// SIMATIC S7-200 SMART project (STEP 7-Micro/WIN SMART), CPU SR40

SYMBOL_TABLE 表格 1
阶段1计数器           C0
阶段2计数器           C1
阶段3计数器           C2
阶段4计数器           C3
阶段5计数器           C4
阶段6计数器           C5
分钟计数器_系统时间       C100
小时计数器_系统时间       C101
轮数计数器_系统时间       C102
通讯状态1            M0.1
通讯状态2            M0.2
本地启动CMD          M2.0
本地停止CMD          M2.1
本地复位CMD          M2.2
远程启动CMD          M3.0
远程停止CMD          M3.1
远程复位CMD          M3.2
PID故障码           MB20
通讯报错1            MB21
通讯报错2            MB22
吹扫时长定时器          T101
点火延时定时器          T102
升降档刷新时间          T103
点失败延时定时器         T104
主火阀开启延时计时器       T105
检漏0延时定时器         T110
检漏1延时定时器         T111
检漏2延时定时器         T112
检漏3延时定时器         T113
检漏4延时定时器         T114
空气阀检测定时器         T115
燃气阀检测定时器         T116
调节阀检测2定时器        T117
DCS安全联锁信号        V0.0
空气压力低检测          V0.1
燃气压力高检测          V0.2
燃气压力低检测          V0.3
JES258故障         V0.4
有火信号             V0.5
启动               V0.6
停止               V0.7
复位               V1.0
本地远程信号           V1.1
故障报警             V2.0
JES运行            V2.1
主火运行             V2.2
故障复位             V2.3
有火指示输出           V2.4
启动状态             V2.5
停止状态             V2.6
安全阀              V2.7
调节阀故障            V3.0
报警显示             V3.1
本地_远程            V20.0
升档               V20.1
降档               V20.2
自动手动             V20.3
PID自动            V20.5
吹扫动画显示           V20.7
无故障点火            V21.0
点火状态             V21.1
开始吹扫             V21.2
开始点火             V21.3
点火成功             V21.4
点火失败             V21.5
火焰信号丢失           V21.6
超温停机             V21.7
燃气阀反馈比对超限        V22.0
空气阀反馈比对超限        V22.1
DCS故障            V22.2
空气压力低            V22.3
燃气压力高            V22.4
燃气压力低            V22.5
空气调节阀故障1         V22.7
燃气调节阀故障          V23.0
调节阀点火位延时         V23.1
吹扫结束             V24.0
点火延时结束           V24.1
故障输出             V24.2
点火延时开始           V24.3
阶段一设定温度读值        V25.0
阶段二设定温度读值        V25.1
条件故障             M4.0
阶段三设定温度读值        V25.2
阶段四设定温度读值        V25.3
阶段五设定温度读值        V25.4
阶段六设定温度读值        V25.5
故障状态RTU          V620.0
自动状态RTU          V620.1
启动状态RTU          V620.2
停止状态RTU          V620.3
远程状态RTU          V620.4
远程启动             V620.5
远程停止             V620.6
远程复位             V620.7
远程升档             V621.0
远程降档             V621.1
当前温度R            VD304
温度显示             VD504
燃气显示             VD508
空气显示             VD512
温度上限设定值          VD520
温度下限设定值          VD524
超温停机设定值          VD528
燃气差              VD532
空气差              VD536
燃气给定             VD540
空气给定             VD544
燃气偏差允许值          VD548
空气偏差允许值          VD552
吹扫空气阀开度          VD564
PID设定温度          VD568
PID微分_D          VD572
PID增益_P          VD576
PID积分_I          VD580
PID采样时间          VD584
PID手动值           VD588
吹扫计时开始_值         VD592
PID档位D           VD596
当前档位显示           VD600
档位设置             VD604
当量_每档            VD608
PID输出换算档位        VD612
PID档位R           VD616
空气               VD640
燃气               VD644
温度               VD648
当前档位             VD652
燃气1档_0档          VD700
燃气2档_点火档         VD704
燃气3档_1档          VD708
燃气4档             VD712
燃气5档             VD716
燃气6档             VD720
燃气7档             VD724
燃气8档             VD728
燃气9档             VD732
燃气10档            VD736
燃气11档            VD740
燃气12档            VD744
燃气13档            VD748
燃气14档            VD752
燃气15档            VD756
燃气16档            VD760
燃气17档            VD764
燃气18档            VD768
燃气19档            VD772
燃气20档            VD776
空气1档             VD780
空气2档             VD784
空气3档             VD788
空气4档             VD792
空气5档             VD796
空气6档             VD800
空气7档             VD804
空气8档             VD808
空气9档             VD812
空气10档            VD816
空气11档            VD820
空气12档            VD824
空气13档            VD828
空气14档            VD832
空气15档            VD836
空气16档            VD840
空气17档            VD844
空气18档            VD848
空气19档            VD852
空气20档            VD856
阶段1温度            VD860
阶段2温度            VD864
阶段3温度            VD868
阶段4温度            VD872
阶段5温度            VD876
阶段6温度            VD880
吹扫时间设定           VW200
点火延时设定值          VW202
吹扫延时             VW206
主火阀开启延时          VW208
PID输出            VW210
阶段1              VW220
阶段2              VW222
阶段3              VW224
阶段4              VW226
阶段5              VW228
阶段6              VW230
阶段1设定            VW232
阶段2设定            VW234
阶段3设定            VW236
阶段4设定            VW238
阶段5设定            VW240
阶段6设定            VW242
调节阀检测延时          VW244
当前温度             VW898
END_SYMBOL_TABLE

SYMBOL_TABLE 系统符号
Always_On        SM0.0    // 始终接通
First_Scan_On    SM0.1    // 仅在第一个扫描周期时接通
Clock_60s        SM0.4    // 针对 1 分钟的周期时间，时钟脉冲接通 30 s，断开 30 s.
Clock_1s         SM0.5    // 针对 1 s 的周期时间，时钟脉冲接通 0.5 s，断开 0.5 s.
END_SYMBOL_TABLE

SYMBOL_TABLE 检漏符号表
检漏标志             VB41     // 0:停止检漏 1:检漏中 2:检漏完成
检漏程序步            VB40     // 检漏第1、2、3、4步
大火指示             V31.0
检漏通过             V30.6
检漏异常2            V30.5
检漏异常1            V30.4
阀1_2             V30.3
阀2_2             V30.2
阀1_1             V30.1
阀2_1             V30.0
检漏异常             V22.6
END_SYMBOL_TABLE

ORGANIZATION_BLOCK 程序块:OB1
TITLE=程序注释
BEGIN
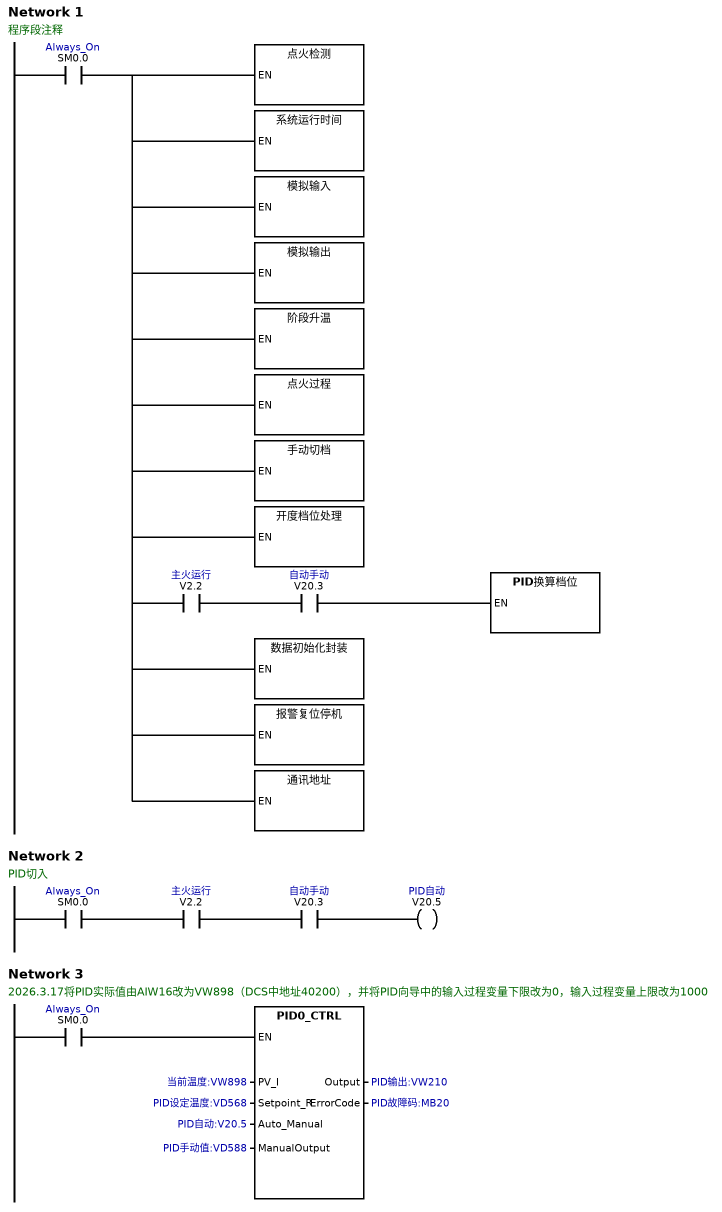
Network 1
// 程序段注释
LD     Always_On:SM0.0
LPS
CALL   点火检测:SBR4
CALL   系统运行时间:SBR5
CALL   模拟输入:SBR0
CALL   模拟输出:SBR3
CALL   阶段升温:SBR6
CALL   点火过程:SBR8
CALL   手动切档:SBR11
CALL   开度档位处理:SBR12
A      主火运行:V2.2
A      自动手动:V20.3
CALL   PID换算档位:SBR13
LRD
CALL   数据初始化封装:SBR14
LRD
CALL   报警复位停机:SBR16
LPP
CALL   通讯地址:SBR19
Network 2
// PID切入
LD     Always_On:SM0.0
A      主火运行:V2.2
A      自动手动:V20.3
=      PID自动:V20.5
Network 3
// 2026.3.17将PID实际值由AIW16改为VW898（DCS中地址40200），并将PID向导中的输入过程变量下限改为0，输入过程变量上限改为1000
LD     Always_On:SM0.0
CALL   PID0_CTRL:SBR18, 当前温度:VW898, PID设定温度:VD568, PID自动:V20.5, PID手动值:VD588, PID输出:VW210, PID故障码:MB20
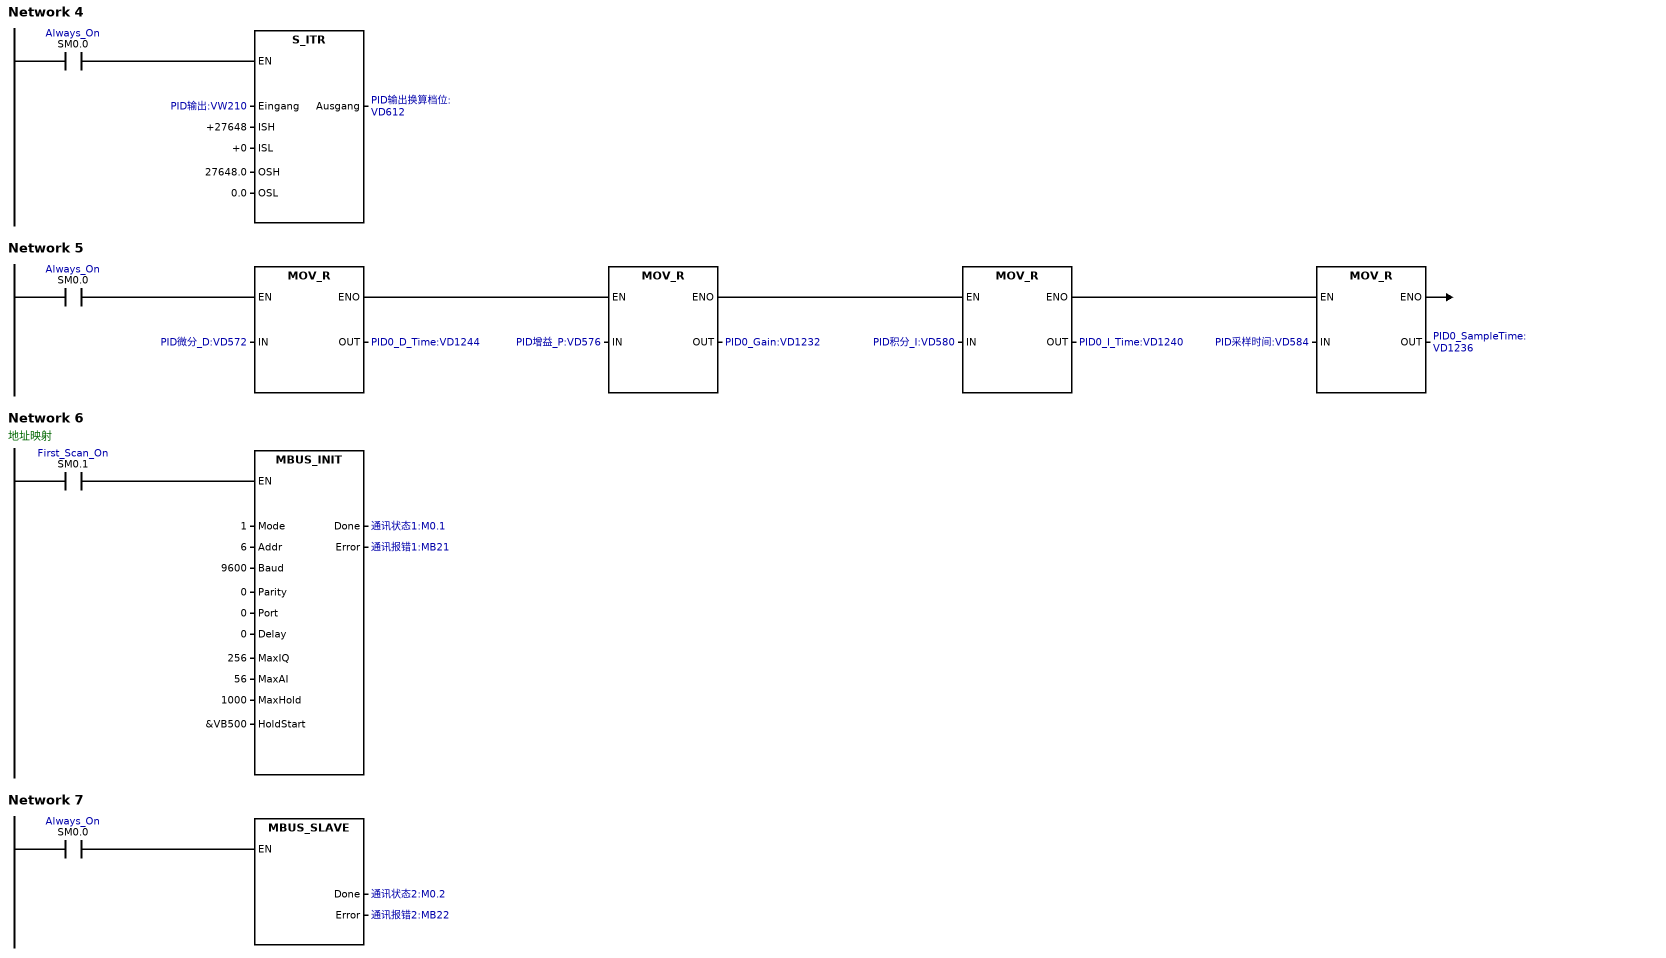
Network 4
LD     Always_On:SM0.0
CALL   S_ITR:SBR1, PID输出:VW210, +27648, +0, 27648.0, 0.0, PID输出换算档位:VD612
Network 5
LD     Always_On:SM0.0
MOVR   PID微分_D:VD572, PID0_D_Time:VD1244
AENO
MOVR   PID增益_P:VD576, PID0_Gain:VD1232
AENO
MOVR   PID积分_I:VD580, PID0_I_Time:VD1240
AENO
MOVR   PID采样时间:VD584, PID0_SampleTime:VD1236
Network 6
// 地址映射
LD     First_Scan_On:SM0.1
CALL   MBUS_INIT:SBR7, 1, 6, 9600, 0, 0, 0, 256, 56, 1000, &VB500, 通讯状态1:M0.1, 通讯报错1:MB21
Network 7
LD     Always_On:SM0.0
CALL   MBUS_SLAVE:SBR9, 通讯状态2:M0.2, 通讯报错2:MB22
END_ORGANIZATION_BLOCK

SUBROUTINE_BLOCK 模拟输入:SBR0
TITLE=子程序注释
BEGIN
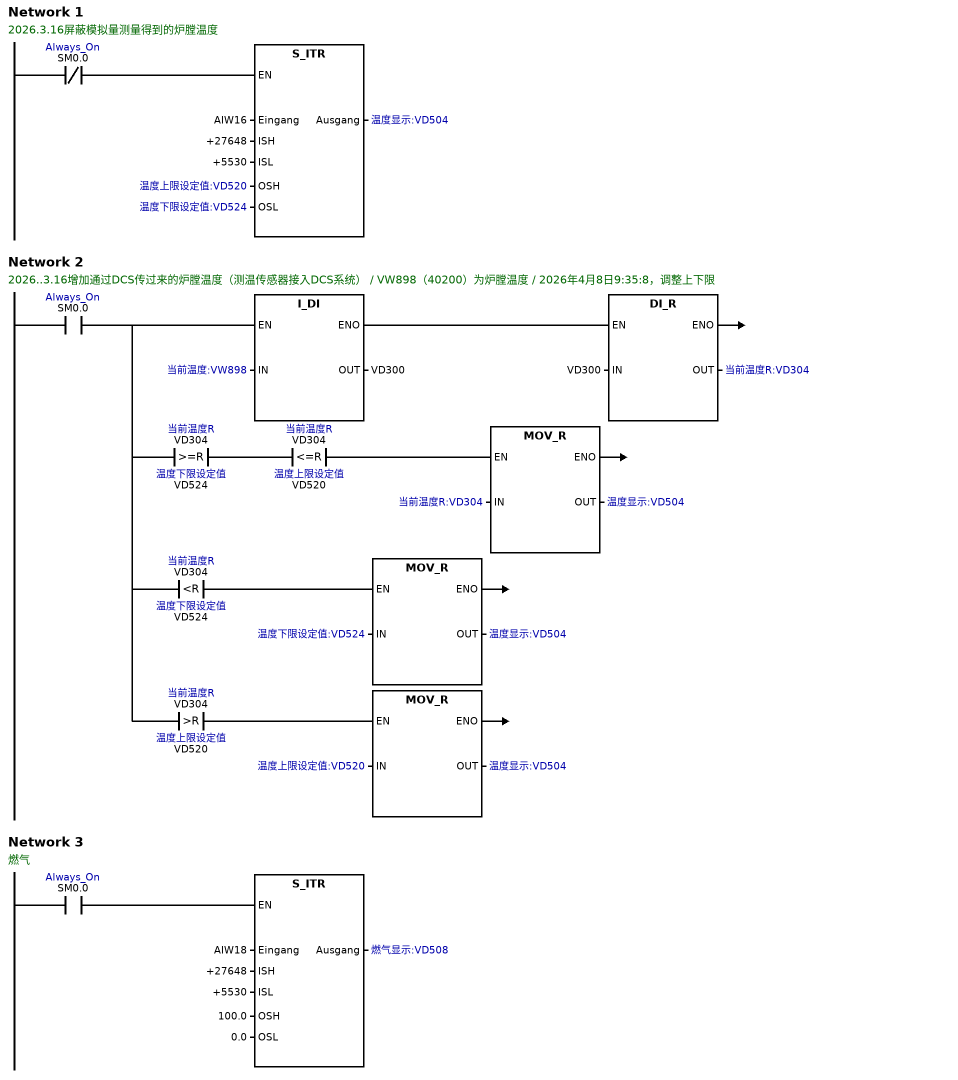
Network 1
// 2026.3.16屏蔽模拟量测量得到的炉膛温度
LDN    Always_On:SM0.0
CALL   S_ITR:SBR1, AIW16, +27648, +5530, 温度上限设定值:VD520, 温度下限设定值:VD524, 温度显示:VD504
Network 2
// 2026..3.16增加通过DCS传过来的炉膛温度（测温传感器接入DCS系统）
// VW898（40200）为炉膛温度
// 2026年4月8日9:35:8，调整上下限
LD     Always_On:SM0.0
LPS
ITD    当前温度:VW898, VD300
AENO
DTR    VD300, 当前温度R:VD304
LRD
AR>=   当前温度R:VD304, 温度下限设定值:VD524
AR<=   当前温度R:VD304, 温度上限设定值:VD520
MOVR   当前温度R:VD304, 温度显示:VD504
LRD
AR<    当前温度R:VD304, 温度下限设定值:VD524
MOVR   温度下限设定值:VD524, 温度显示:VD504
LPP
AR>    当前温度R:VD304, 温度上限设定值:VD520
MOVR   温度上限设定值:VD520, 温度显示:VD504
Network 3
// 燃气
LD     Always_On:SM0.0
CALL   S_ITR:SBR1, AIW18, +27648, +5530, 100.0, 0.0, 燃气显示:VD508
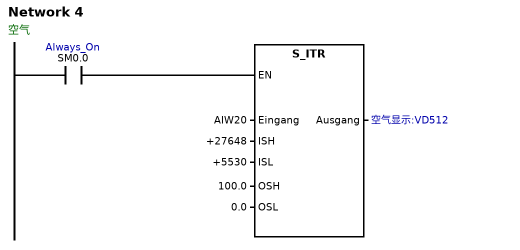
Network 4
// 空气
LD     Always_On:SM0.0
CALL   S_ITR:SBR1, AIW20, +27648, +5530, 100.0, 0.0, 空气显示:VD512
END_SUBROUTINE_BLOCK

// SBR1: protected block, not included

// SBR2: protected block, not included

SUBROUTINE_BLOCK 模拟输出:SBR3
TITLE=
BEGIN
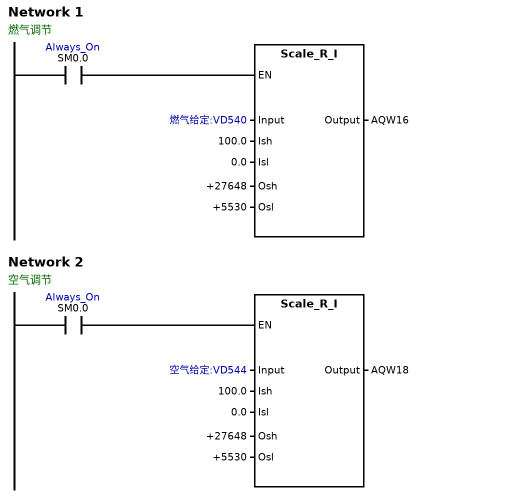
Network 1
// 燃气调节
LD     Always_On:SM0.0
CALL   Scale_R_I:SBR17, 燃气给定:VD540, 100.0, 0.0, +27648, +5530, AQW16
Network 2
// 空气调节
LD     Always_On:SM0.0
CALL   Scale_R_I:SBR17, 空气给定:VD544, 100.0, 0.0, +27648, +5530, AQW18
END_SUBROUTINE_BLOCK

SUBROUTINE_BLOCK 点火检测:SBR4
TITLE=
BEGIN
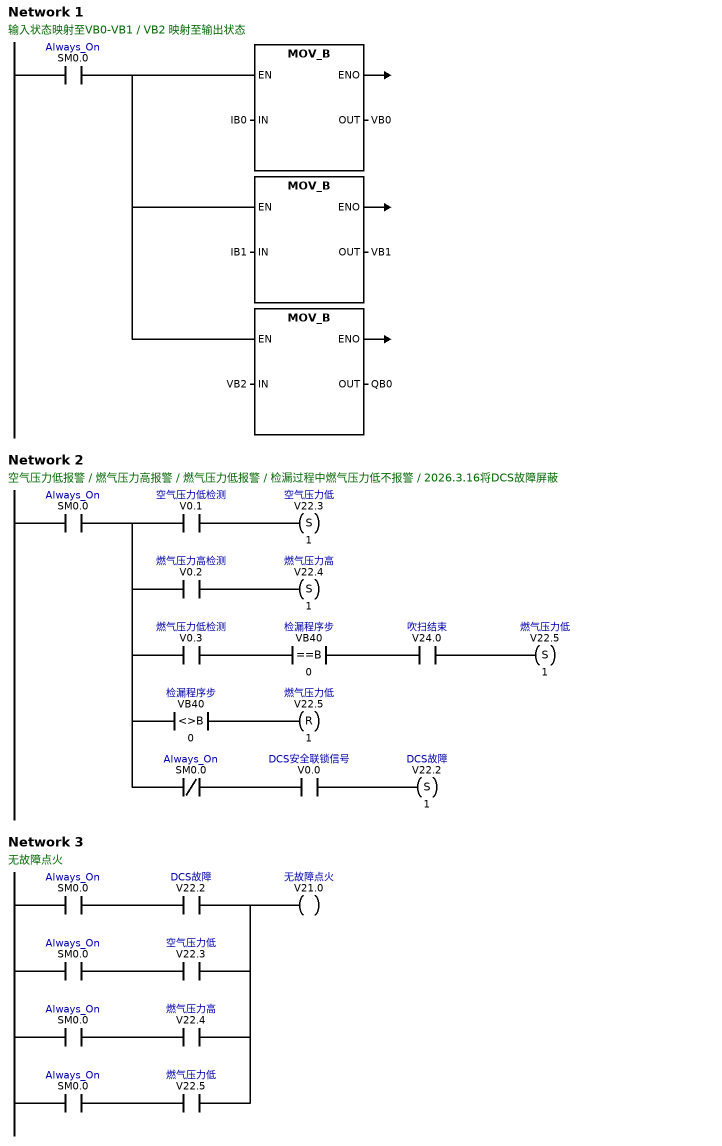
Network 1
// 输入状态映射至VB0-VB1
// VB2 映射至输出状态
LD     Always_On:SM0.0
MOVB   IB0, VB0
MOVB   IB1, VB1
MOVB   VB2, QB0
Network 2
// 空气压力低报警
// 燃气压力高报警
// 燃气压力低报警
// 检漏过程中燃气压力低不报警
// 2026.3.16将DCS故障屏蔽
LD     Always_On:SM0.0
LPS
A      空气压力低检测:V0.1
S      空气压力低:V22.3, 1
LRD
A      燃气压力高检测:V0.2
S      燃气压力高:V22.4, 1
LRD
A      燃气压力低检测:V0.3
AB=    检漏程序步:VB40, 0
A      吹扫结束:V24.0
S      燃气压力低:V22.5, 1
LRD
AB<>   检漏程序步:VB40, 0
R      燃气压力低:V22.5, 1
LPP
AN     Always_On:SM0.0
A      DCS安全联锁信号:V0.0
S      DCS故障:V22.2, 1
Network 3
// 无故障点火
LD     Always_On:SM0.0
A      DCS故障:V22.2
LD     Always_On:SM0.0
A      空气压力低:V22.3
OLD
LD     Always_On:SM0.0
A      燃气压力高:V22.4
OLD
LD     Always_On:SM0.0
A      燃气压力低:V22.5
OLD
=      无故障点火:V21.0
END_SUBROUTINE_BLOCK

SUBROUTINE_BLOCK 系统运行时间:SBR5
TITLE=
BEGIN
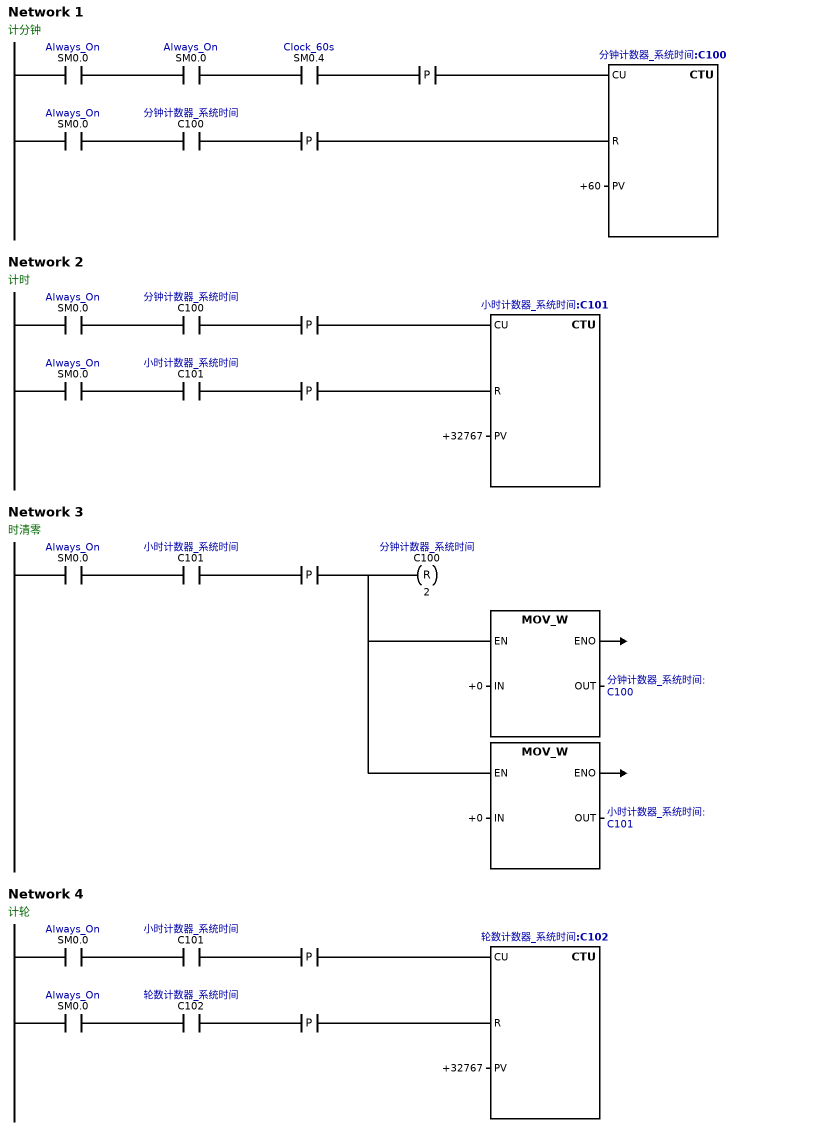
Network 1
// 计分钟
LD     Always_On:SM0.0
A      Always_On:SM0.0
A      Clock_60s:SM0.4
EU
LD     Always_On:SM0.0
A      分钟计数器_系统时间:C100
EU
CTU    分钟计数器_系统时间:C100, +60
Network 2
// 计时
LD     Always_On:SM0.0
A      分钟计数器_系统时间:C100
EU
LD     Always_On:SM0.0
A      小时计数器_系统时间:C101
EU
CTU    小时计数器_系统时间:C101, +32767
Network 3
// 时清零
LD     Always_On:SM0.0
A      小时计数器_系统时间:C101
EU
R      分钟计数器_系统时间:C100, 2
MOVW   +0, 分钟计数器_系统时间:C100
MOVW   +0, 小时计数器_系统时间:C101
Network 4
// 计轮
LD     Always_On:SM0.0
A      小时计数器_系统时间:C101
EU
LD     Always_On:SM0.0
A      轮数计数器_系统时间:C102
EU
CTU    轮数计数器_系统时间:C102, +32767
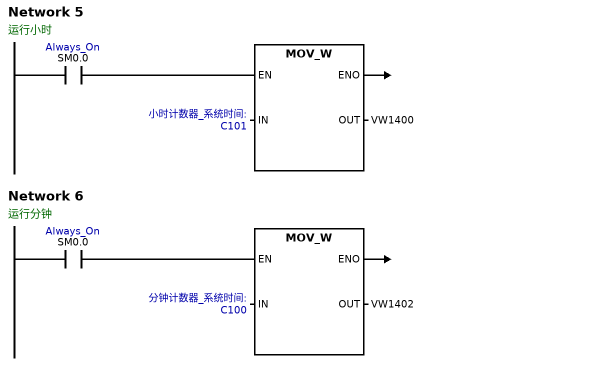
Network 5
// 运行小时
LD     Always_On:SM0.0
MOVW   小时计数器_系统时间:C101, VW1400
Network 6
// 运行分钟
LD     Always_On:SM0.0
MOVW   分钟计数器_系统时间:C100, VW1402
END_SUBROUTINE_BLOCK

SUBROUTINE_BLOCK 阶段升温:SBR6
TITLE=
BEGIN
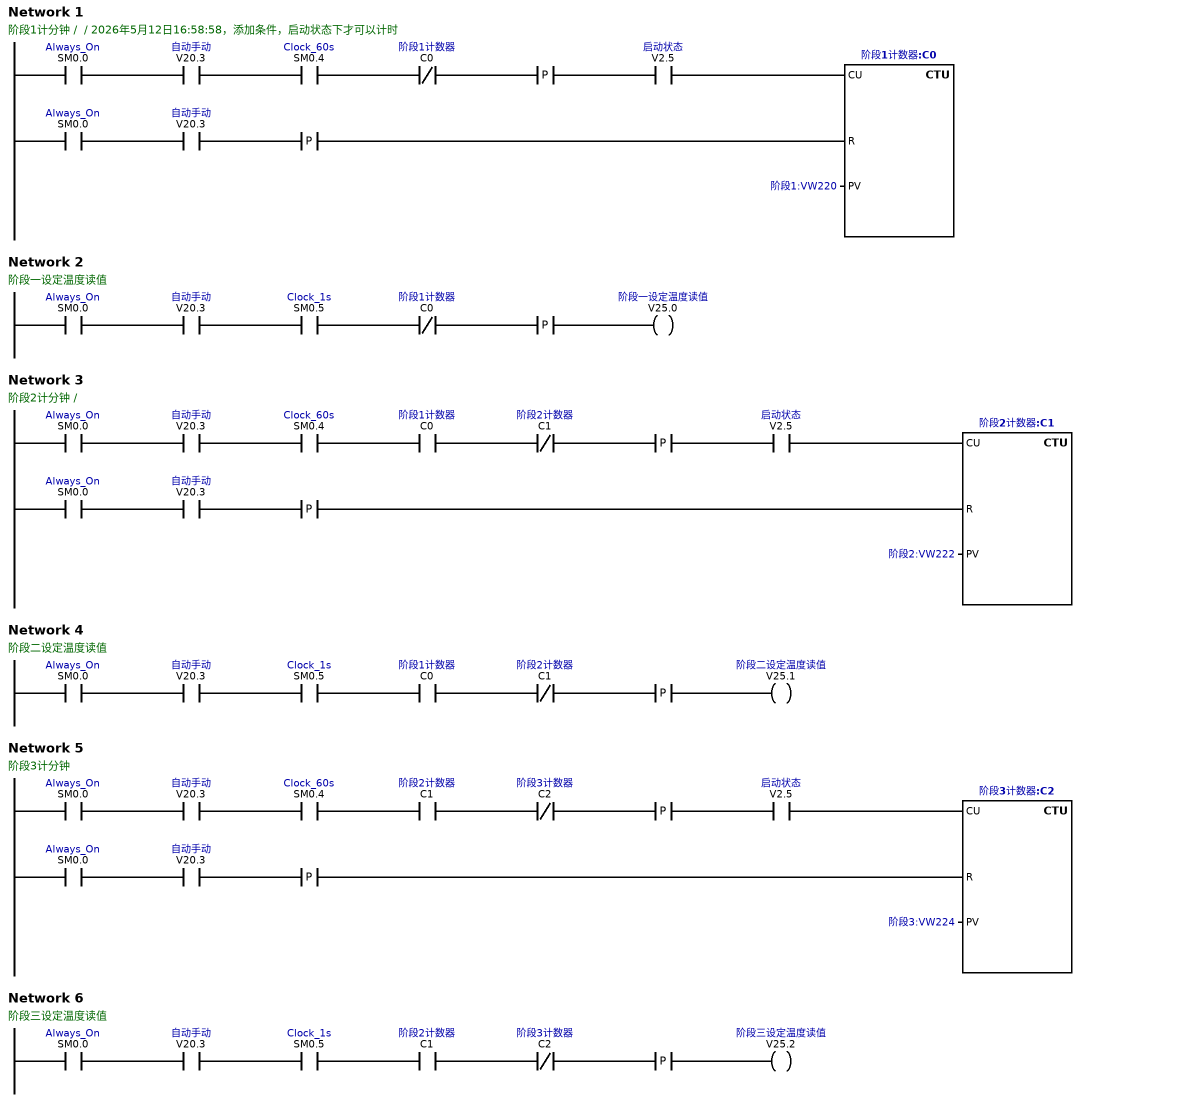
Network 1
// 阶段1计分钟
// 
// 2026年5月12日16:58:58，添加条件，启动状态下才可以计时
LD     Always_On:SM0.0
A      自动手动:V20.3
A      Clock_60s:SM0.4
AN     阶段1计数器:C0
EU
A      启动状态:V2.5
LD     Always_On:SM0.0
A      自动手动:V20.3
EU
CTU    阶段1计数器:C0, 阶段1:VW220
Network 2
// 阶段一设定温度读值
LD     Always_On:SM0.0
A      自动手动:V20.3
A      Clock_1s:SM0.5
AN     阶段1计数器:C0
EU
=      阶段一设定温度读值:V25.0
Network 3
// 阶段2计分钟
// 
LD     Always_On:SM0.0
A      自动手动:V20.3
A      Clock_60s:SM0.4
A      阶段1计数器:C0
AN     阶段2计数器:C1
EU
A      启动状态:V2.5
LD     Always_On:SM0.0
A      自动手动:V20.3
EU
CTU    阶段2计数器:C1, 阶段2:VW222
Network 4
// 阶段二设定温度读值
LD     Always_On:SM0.0
A      自动手动:V20.3
A      Clock_1s:SM0.5
A      阶段1计数器:C0
AN     阶段2计数器:C1
EU
=      阶段二设定温度读值:V25.1
Network 5
// 阶段3计分钟
LD     Always_On:SM0.0
A      自动手动:V20.3
A      Clock_60s:SM0.4
A      阶段2计数器:C1
AN     阶段3计数器:C2
EU
A      启动状态:V2.5
LD     Always_On:SM0.0
A      自动手动:V20.3
EU
CTU    阶段3计数器:C2, 阶段3:VW224
Network 6
// 阶段三设定温度读值
LD     Always_On:SM0.0
A      自动手动:V20.3
A      Clock_1s:SM0.5
A      阶段2计数器:C1
AN     阶段3计数器:C2
EU
=      阶段三设定温度读值:V25.2
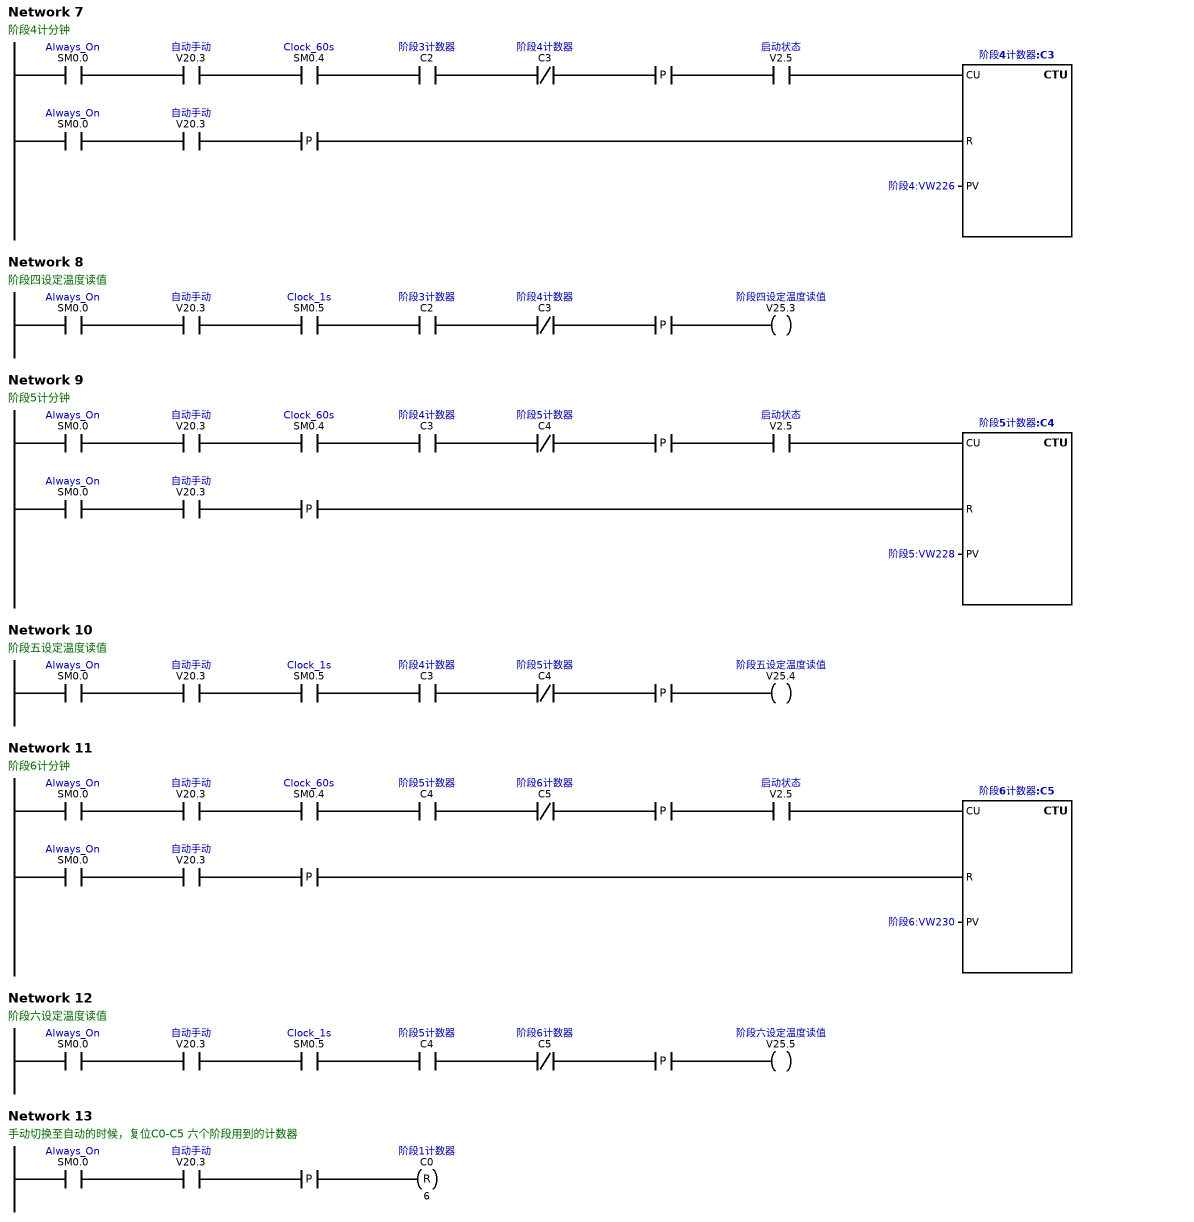
Network 7
// 阶段4计分钟
LD     Always_On:SM0.0
A      自动手动:V20.3
A      Clock_60s:SM0.4
A      阶段3计数器:C2
AN     阶段4计数器:C3
EU
A      启动状态:V2.5
LD     Always_On:SM0.0
A      自动手动:V20.3
EU
CTU    阶段4计数器:C3, 阶段4:VW226
Network 8
// 阶段四设定温度读值
LD     Always_On:SM0.0
A      自动手动:V20.3
A      Clock_1s:SM0.5
A      阶段3计数器:C2
AN     阶段4计数器:C3
EU
=      阶段四设定温度读值:V25.3
Network 9
// 阶段5计分钟
LD     Always_On:SM0.0
A      自动手动:V20.3
A      Clock_60s:SM0.4
A      阶段4计数器:C3
AN     阶段5计数器:C4
EU
A      启动状态:V2.5
LD     Always_On:SM0.0
A      自动手动:V20.3
EU
CTU    阶段5计数器:C4, 阶段5:VW228
Network 10
// 阶段五设定温度读值
LD     Always_On:SM0.0
A      自动手动:V20.3
A      Clock_1s:SM0.5
A      阶段4计数器:C3
AN     阶段5计数器:C4
EU
=      阶段五设定温度读值:V25.4
Network 11
// 阶段6计分钟
LD     Always_On:SM0.0
A      自动手动:V20.3
A      Clock_60s:SM0.4
A      阶段5计数器:C4
AN     阶段6计数器:C5
EU
A      启动状态:V2.5
LD     Always_On:SM0.0
A      自动手动:V20.3
EU
CTU    阶段6计数器:C5, 阶段6:VW230
Network 12
// 阶段六设定温度读值
LD     Always_On:SM0.0
A      自动手动:V20.3
A      Clock_1s:SM0.5
A      阶段5计数器:C4
AN     阶段6计数器:C5
EU
=      阶段六设定温度读值:V25.5
Network 13
// 手动切换至自动的时候，复位C0-C5 六个阶段用到的计数器
LD     Always_On:SM0.0
A      自动手动:V20.3
EU
R      阶段1计数器:C0, 6
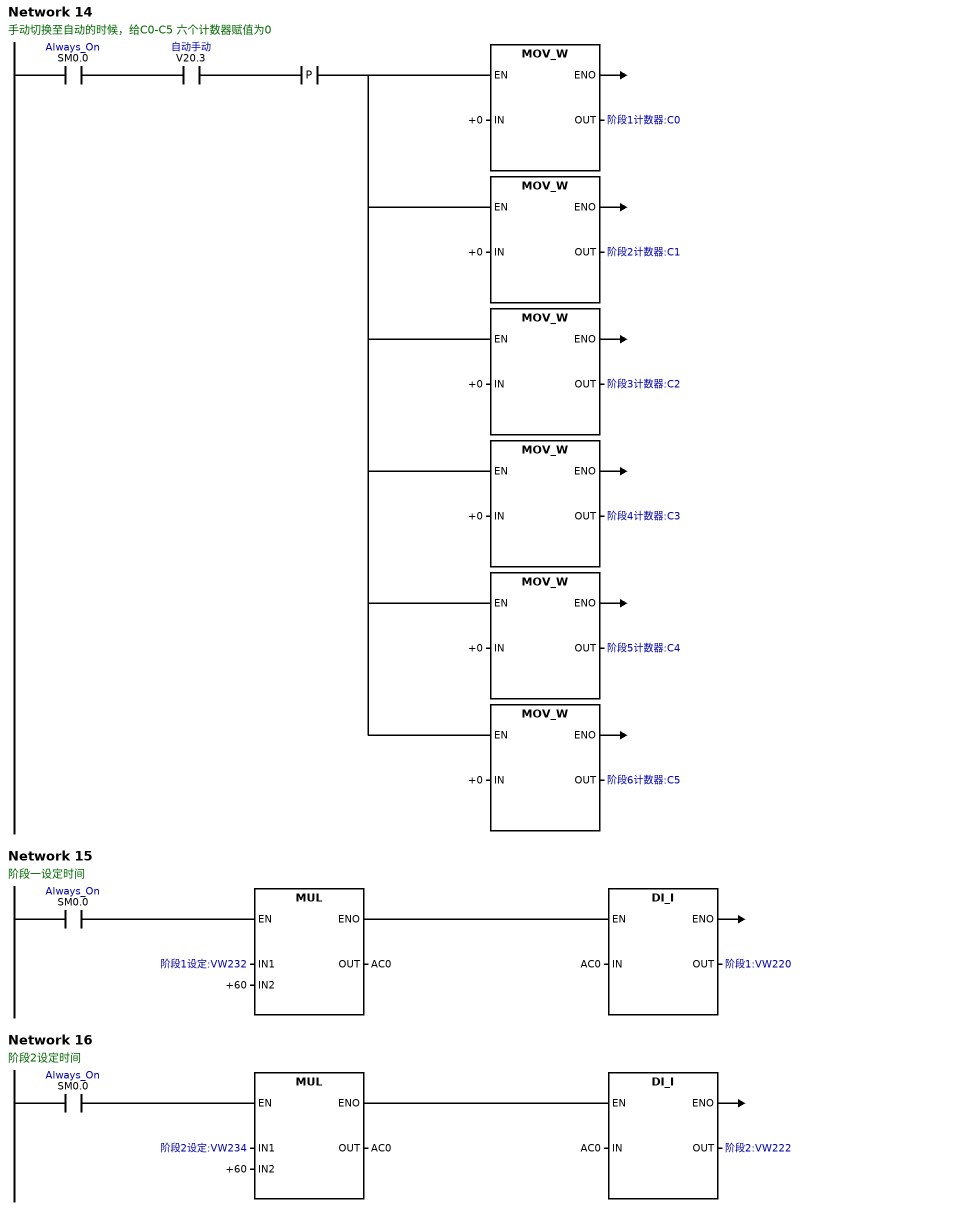
Network 14
// 手动切换至自动的时候，给C0-C5 六个计数器赋值为0
LD     Always_On:SM0.0
A      自动手动:V20.3
EU
MOVW   +0, 阶段1计数器:C0
MOVW   +0, 阶段2计数器:C1
MOVW   +0, 阶段3计数器:C2
MOVW   +0, 阶段4计数器:C3
MOVW   +0, 阶段5计数器:C4
MOVW   +0, 阶段6计数器:C5
Network 15
// 阶段一设定时间
LD     Always_On:SM0.0
MOVW   阶段1设定:VW232, AC0
AENO
MUL    +60, AC0
AENO
DTI    AC0, 阶段1:VW220
Network 16
// 阶段2设定时间
LD     Always_On:SM0.0
MOVW   阶段2设定:VW234, AC0
AENO
MUL    +60, AC0
AENO
DTI    AC0, 阶段2:VW222
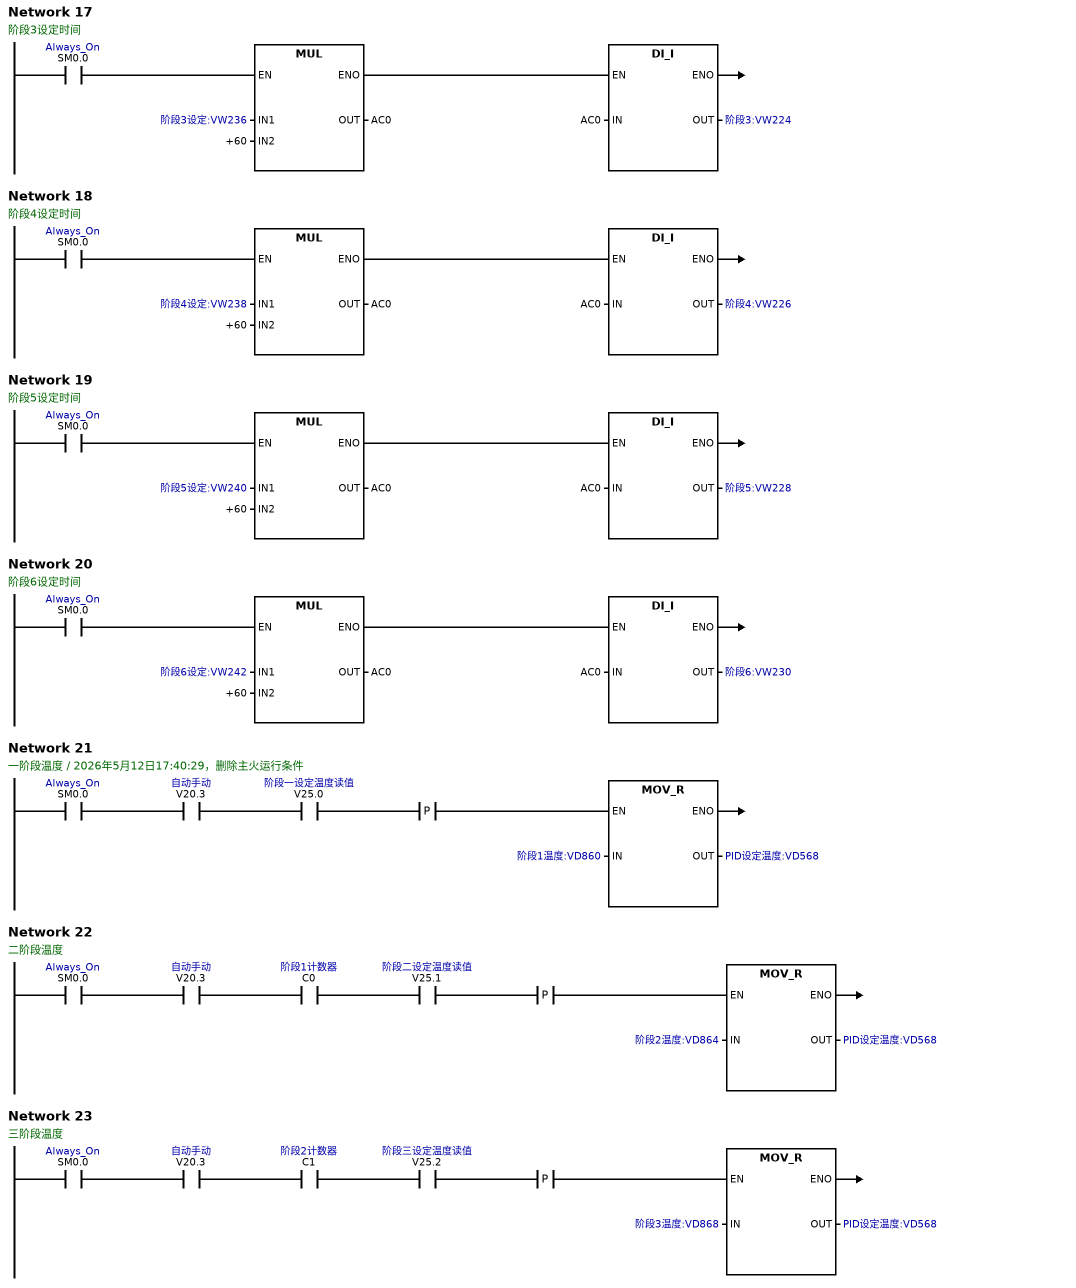
Network 17
// 阶段3设定时间
LD     Always_On:SM0.0
MOVW   阶段3设定:VW236, AC0
AENO
MUL    +60, AC0
AENO
DTI    AC0, 阶段3:VW224
Network 18
// 阶段4设定时间
LD     Always_On:SM0.0
MOVW   阶段4设定:VW238, AC0
AENO
MUL    +60, AC0
AENO
DTI    AC0, 阶段4:VW226
Network 19
// 阶段5设定时间
LD     Always_On:SM0.0
MOVW   阶段5设定:VW240, AC0
AENO
MUL    +60, AC0
AENO
DTI    AC0, 阶段5:VW228
Network 20
// 阶段6设定时间
LD     Always_On:SM0.0
MOVW   阶段6设定:VW242, AC0
AENO
MUL    +60, AC0
AENO
DTI    AC0, 阶段6:VW230
Network 21
// 一阶段温度
// 2026年5月12日17:40:29，删除主火运行条件
LD     Always_On:SM0.0
A      自动手动:V20.3
A      阶段一设定温度读值:V25.0
EU
MOVR   阶段1温度:VD860, PID设定温度:VD568
Network 22
// 二阶段温度
LD     Always_On:SM0.0
A      自动手动:V20.3
A      阶段1计数器:C0
A      阶段二设定温度读值:V25.1
EU
MOVR   阶段2温度:VD864, PID设定温度:VD568
Network 23
// 三阶段温度
LD     Always_On:SM0.0
A      自动手动:V20.3
A      阶段2计数器:C1
A      阶段三设定温度读值:V25.2
EU
MOVR   阶段3温度:VD868, PID设定温度:VD568
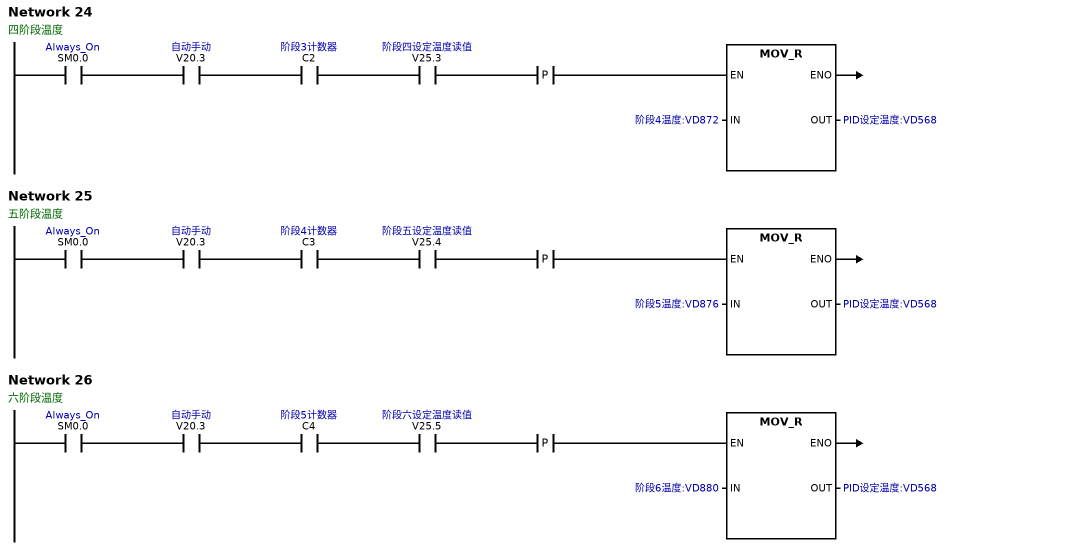
Network 24
// 四阶段温度
LD     Always_On:SM0.0
A      自动手动:V20.3
A      阶段3计数器:C2
A      阶段四设定温度读值:V25.3
EU
MOVR   阶段4温度:VD872, PID设定温度:VD568
Network 25
// 五阶段温度
LD     Always_On:SM0.0
A      自动手动:V20.3
A      阶段4计数器:C3
A      阶段五设定温度读值:V25.4
EU
MOVR   阶段5温度:VD876, PID设定温度:VD568
Network 26
// 六阶段温度
LD     Always_On:SM0.0
A      自动手动:V20.3
A      阶段5计数器:C4
A      阶段六设定温度读值:V25.5
EU
MOVR   阶段6温度:VD880, PID设定温度:VD568
END_SUBROUTINE_BLOCK

// SBR7: protected block, not included

SUBROUTINE_BLOCK 点火过程:SBR8
TITLE=
BEGIN
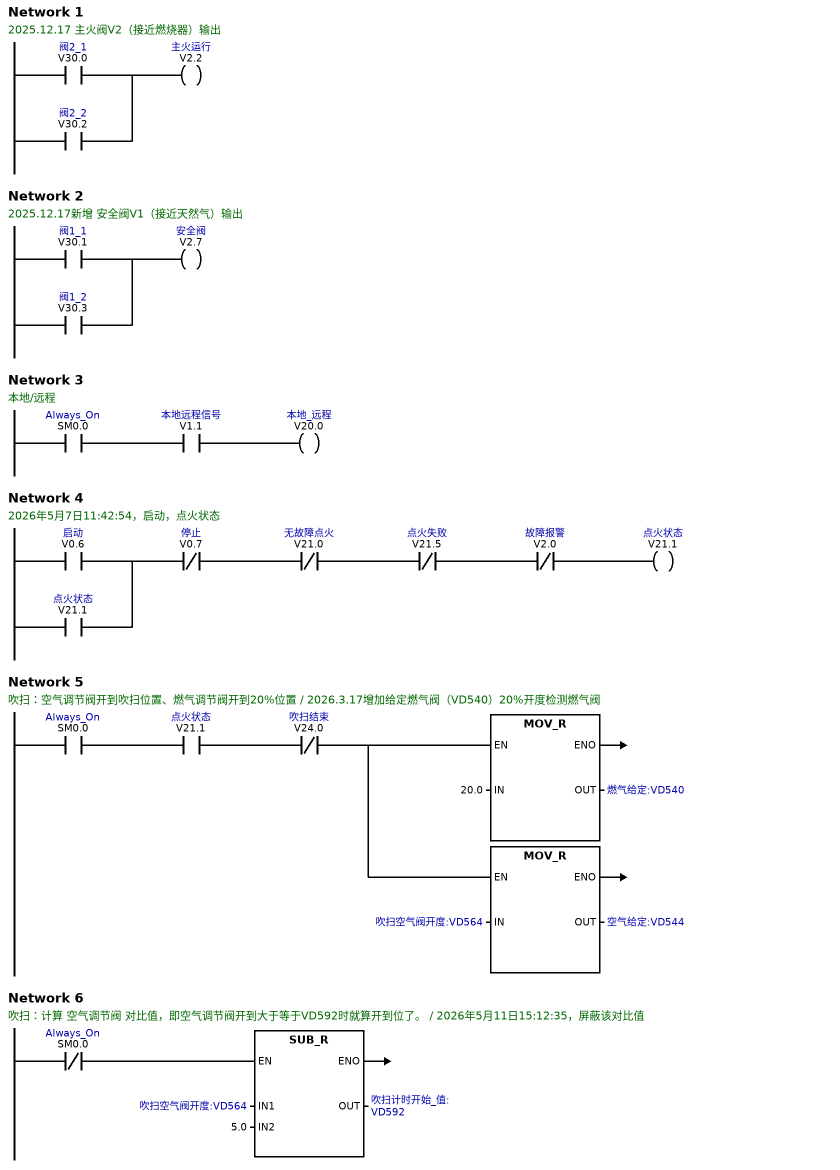
Network 1
// 2025.12.17 主火阀V2（接近燃烧器）输出
LD     阀2_1:V30.0
O      阀2_2:V30.2
=      主火运行:V2.2
Network 2
// 2025.12.17新增 安全阀V1（接近天然气）输出
LD     阀1_1:V30.1
O      阀1_2:V30.3
=      安全阀:V2.7
Network 3
// 本地/远程
LD     Always_On:SM0.0
A      本地远程信号:V1.1
=      本地_远程:V20.0
Network 4
// 2026年5月7日11:42:54，启动，点火状态
LD     启动:V0.6
O      点火状态:V21.1
AN     停止:V0.7
AN     无故障点火:V21.0
AN     点火失败:V21.5
AN     故障报警:V2.0
=      点火状态:V21.1
Network 5
// 吹扫：空气调节阀开到吹扫位置、燃气调节阀开到20%位置
// 2026.3.17增加给定燃气阀（VD540）20%开度检测燃气阀
LD     Always_On:SM0.0
A      点火状态:V21.1
AN     吹扫结束:V24.0
MOVR   20.0, 燃气给定:VD540
MOVR   吹扫空气阀开度:VD564, 空气给定:VD544
Network 6
// 吹扫：计算 空气调节阀 对比值，即空气调节阀开到大于等于VD592时就算开到位了。
// 2026年5月11日15:12:35，屏蔽该对比值
LDN    Always_On:SM0.0
MOVR   吹扫空气阀开度:VD564, 吹扫计时开始_值:VD592
-R     5.0, 吹扫计时开始_值:VD592
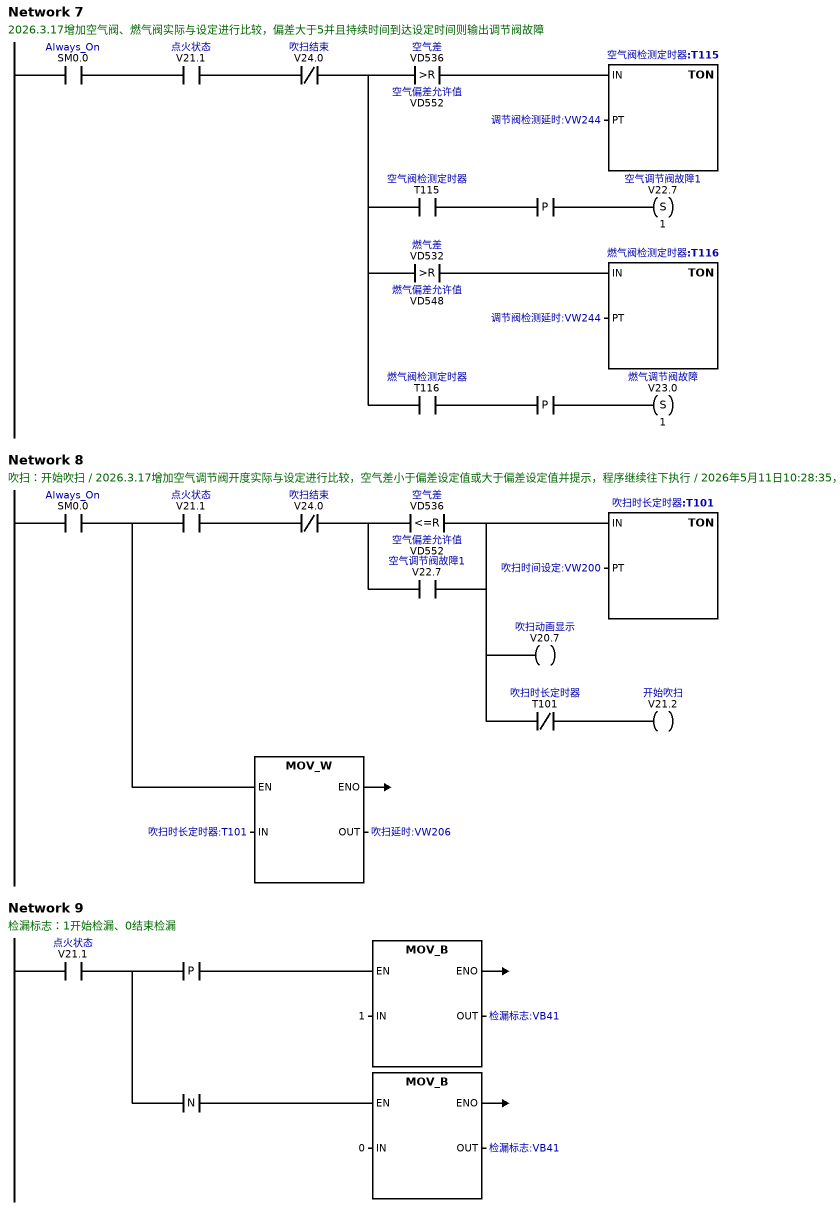
Network 7
// 2026.3.17增加空气阀、燃气阀实际与设定进行比较，偏差大于5并且持续时间到达设定时间则输出调节阀故障
LD     Always_On:SM0.0
A      点火状态:V21.1
AN     吹扫结束:V24.0
LPS
AR>    空气差:VD536, 空气偏差允许值:VD552
TON    空气阀检测定时器:T115, 调节阀检测延时:VW244
LRD
A      空气阀检测定时器:T115
EU
S      空气调节阀故障1:V22.7, 1
LRD
AR>    燃气差:VD532, 燃气偏差允许值:VD548
TON    燃气阀检测定时器:T116, 调节阀检测延时:VW244
LPP
A      燃气阀检测定时器:T116
EU
S      燃气调节阀故障:V23.0, 1
Network 8
// 吹扫：开始吹扫
// 2026.3.17增加空气调节阀开度实际与设定进行比较，空气差小于偏差设定值或大于偏差设定值并提示，程序继续往下执行
// 2026年5月11日10:28:35，显示吹扫时长
LD     Always_On:SM0.0
LPS
A      点火状态:V21.1
AN     吹扫结束:V24.0
LDR<=  空气差:VD536, 空气偏差允许值:VD552
O      空气调节阀故障1:V22.7
ALD
TON    吹扫时长定时器:T101, 吹扫时间设定:VW200
=      吹扫动画显示:V20.7
AN     吹扫时长定时器:T101
=      开始吹扫:V21.2
LPP
MOVW   吹扫时长定时器:T101, 吹扫延时:VW206
Network 9
// 检漏标志：1开始检漏、0结束检漏
LD     点火状态:V21.1
LPS
EU
MOVB   1, 检漏标志:VB41
LPP
ED
MOVB   0, 检漏标志:VB41
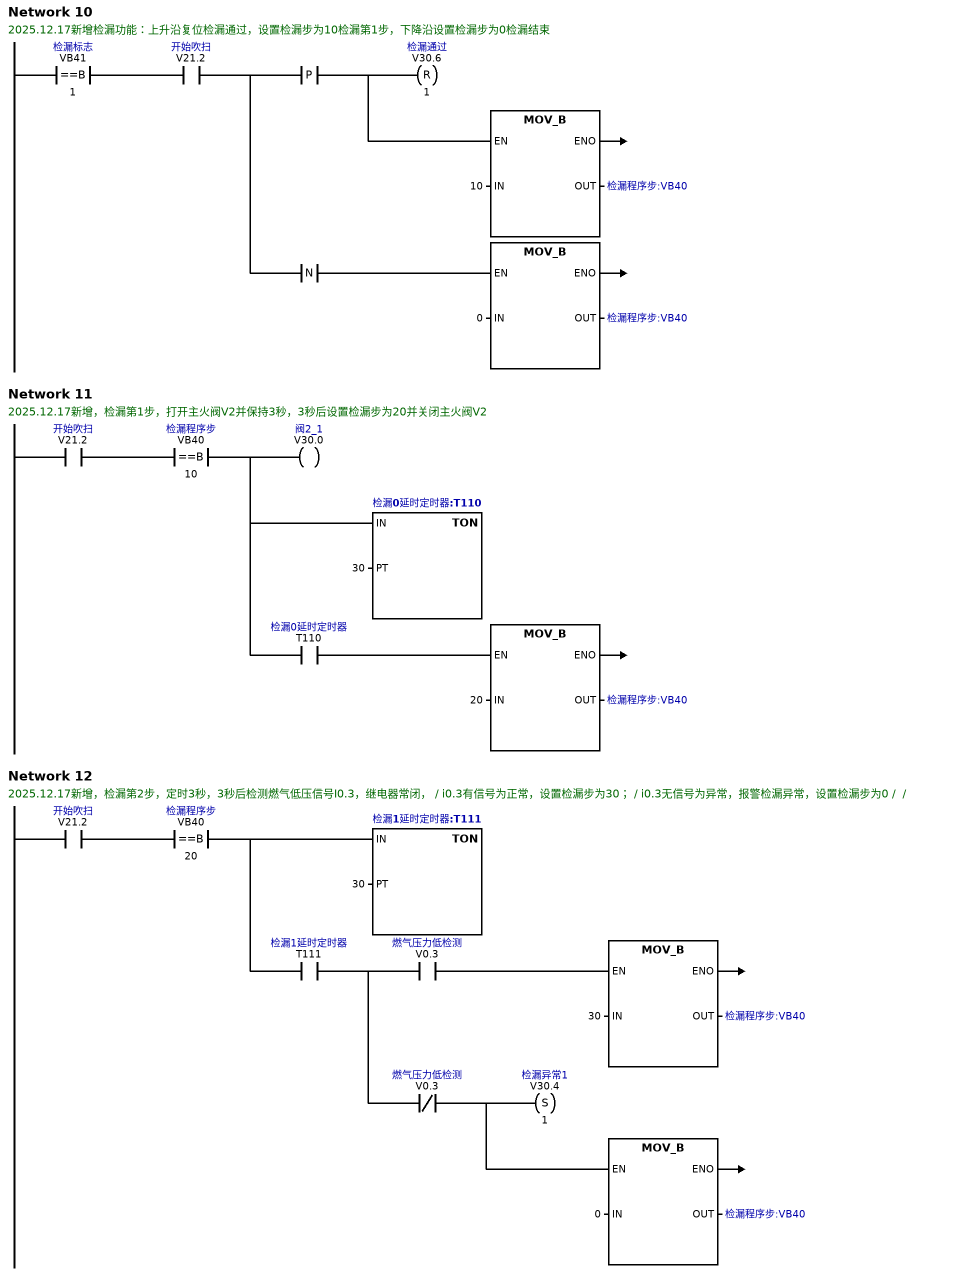
Network 10
// 2025.12.17新增检漏功能：上升沿复位检漏通过，设置检漏步为10检漏第1步，下降沿设置检漏步为0检漏结束
LDB=   检漏标志:VB41, 1
A      开始吹扫:V21.2
LPS
EU
R      检漏通过:V30.6, 1
MOVB   10, 检漏程序步:VB40
LPP
ED
MOVB   0, 检漏程序步:VB40
Network 11
// 2025.12.17新增，检漏第1步，打开主火阀V2并保持3秒，3秒后设置检漏步为20并关闭主火阀V2
LD     开始吹扫:V21.2
AB=    检漏程序步:VB40, 10
=      阀2_1:V30.0
TON    检漏0延时定时器:T110, 30
A      检漏0延时定时器:T110
MOVB   20, 检漏程序步:VB40
Network 12
// 2025.12.17新增，检漏第2步，定时3秒，3秒后检测燃气低压信号I0.3，继电器常闭，
// i0.3有信号为正常，设置检漏步为30；
// i0.3无信号为异常，报警检漏异常，设置检漏步为0
// 
// 
LD     开始吹扫:V21.2
AB=    检漏程序步:VB40, 20
TON    检漏1延时定时器:T111, 30
A      检漏1延时定时器:T111
LPS
A      燃气压力低检测:V0.3
MOVB   30, 检漏程序步:VB40
LPP
AN     燃气压力低检测:V0.3
S      检漏异常1:V30.4, 1
MOVB   0, 检漏程序步:VB40
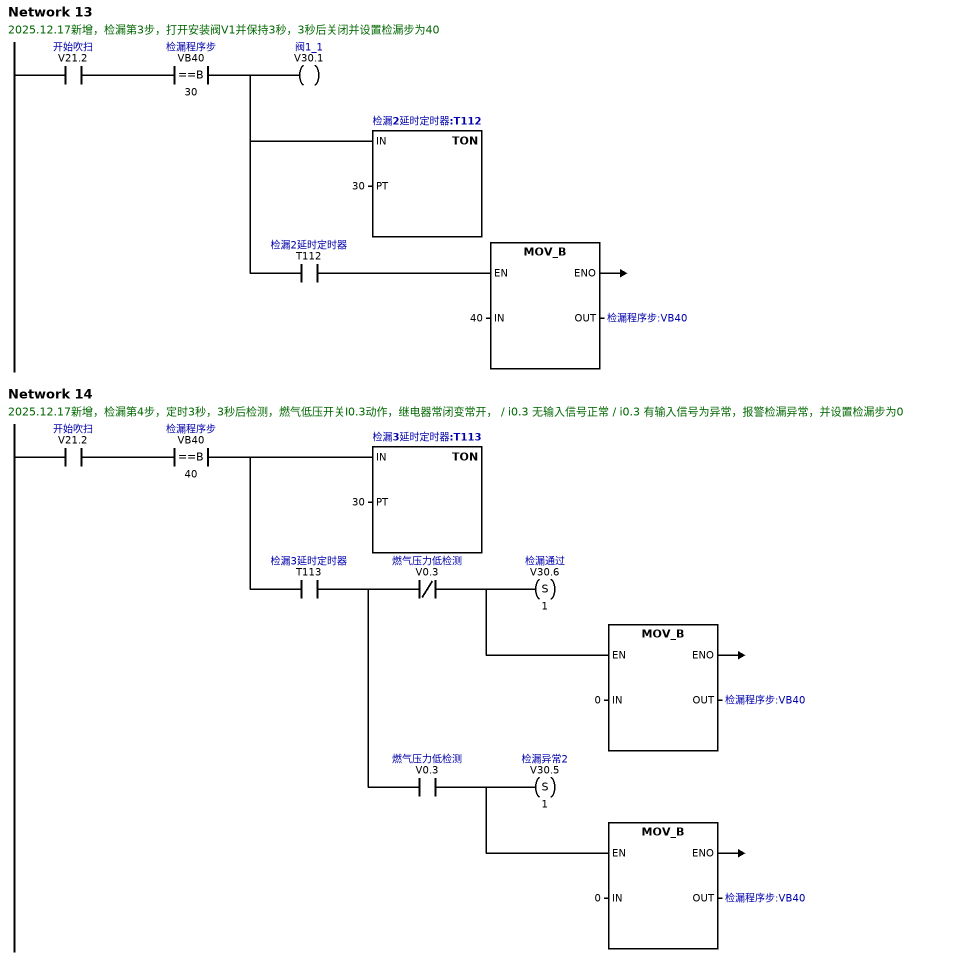
Network 13
// 2025.12.17新增，检漏第3步，打开安装阀V1并保持3秒，3秒后关闭并设置检漏步为40
LD     开始吹扫:V21.2
AB=    检漏程序步:VB40, 30
=      阀1_1:V30.1
TON    检漏2延时定时器:T112, 30
A      检漏2延时定时器:T112
MOVB   40, 检漏程序步:VB40
Network 14
// 2025.12.17新增，检漏第4步，定时3秒，3秒后检测，燃气低压开关I0.3动作，继电器常闭变常开，
// i0.3 无输入信号正常
// i0.3 有输入信号为异常，报警检漏异常，并设置检漏步为0
LD     开始吹扫:V21.2
AB=    检漏程序步:VB40, 40
TON    检漏3延时定时器:T113, 30
A      检漏3延时定时器:T113
LPS
AN     燃气压力低检测:V0.3
S      检漏通过:V30.6, 1
MOVB   0, 检漏程序步:VB40
LPP
A      燃气压力低检测:V0.3
S      检漏异常2:V30.5, 1
MOVB   0, 检漏程序步:VB40
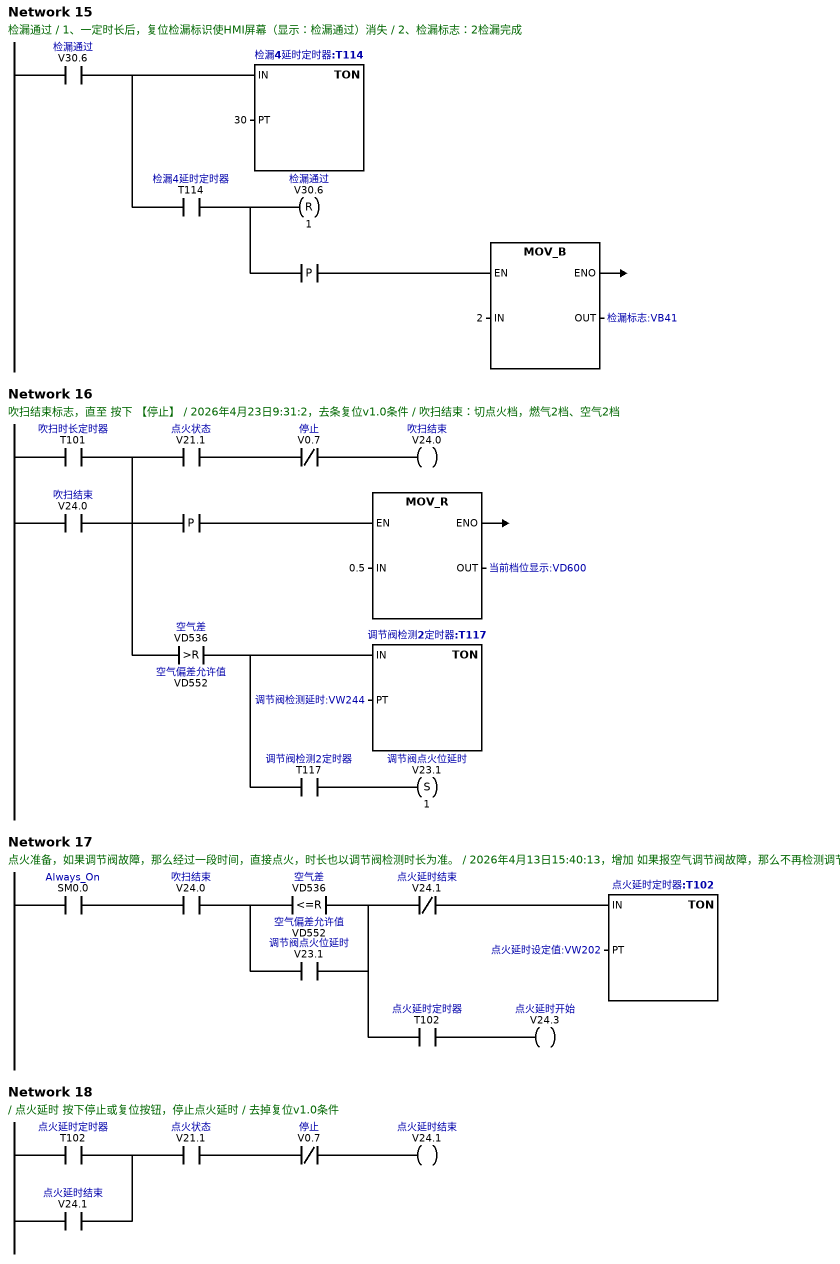
Network 15
// 检漏通过
// 1、一定时长后，复位检漏标识使HMI屏幕（显示：检漏通过）消失
// 2、检漏标志：2检漏完成
LD     检漏通过:V30.6
TON    检漏4延时定时器:T114, 30
A      检漏4延时定时器:T114
R      检漏通过:V30.6, 1
EU
MOVB   2, 检漏标志:VB41
Network 16
// 吹扫结束标志，直至 按下 【停止】
// 2026年4月23日9:31:2，去条复位v1.0条件
// 吹扫结束：切点火档，燃气2档、空气2档
LD     吹扫时长定时器:T101
O      吹扫结束:V24.0
LPS
A      点火状态:V21.1
AN     停止:V0.7
=      吹扫结束:V24.0
LRD
EU
MOVR   0.5, 当前档位显示:VD600
LPP
AR>    空气差:VD536, 空气偏差允许值:VD552
TON    调节阀检测2定时器:T117, 调节阀检测延时:VW244
A      调节阀检测2定时器:T117
S      调节阀点火位延时:V23.1, 1
Network 17
// 点火准备，如果调节阀故障，那么经过一段时间，直接点火，时长也以调节阀检测时长为准。
// 2026年4月13日15:40:13，增加 如果报空气调节阀故障，那么不再检测调节阀，一定时长后继续往下运行程序。
LD     Always_On:SM0.0
A      吹扫结束:V24.0
LDR<=  空气差:VD536, 空气偏差允许值:VD552
O      调节阀点火位延时:V23.1
ALD
LPS
AN     点火延时结束:V24.1
TON    点火延时定时器:T102, 点火延时设定值:VW202
LPP
A      点火延时定时器:T102
=      点火延时开始:V24.3
Network 18
// 
// 点火延时 按下停止或复位按钮，停止点火延时
// 去掉复位v1.0条件
LD     点火延时定时器:T102
O      点火延时结束:V24.1
A      点火状态:V21.1
AN     停止:V0.7
=      点火延时结束:V24.1
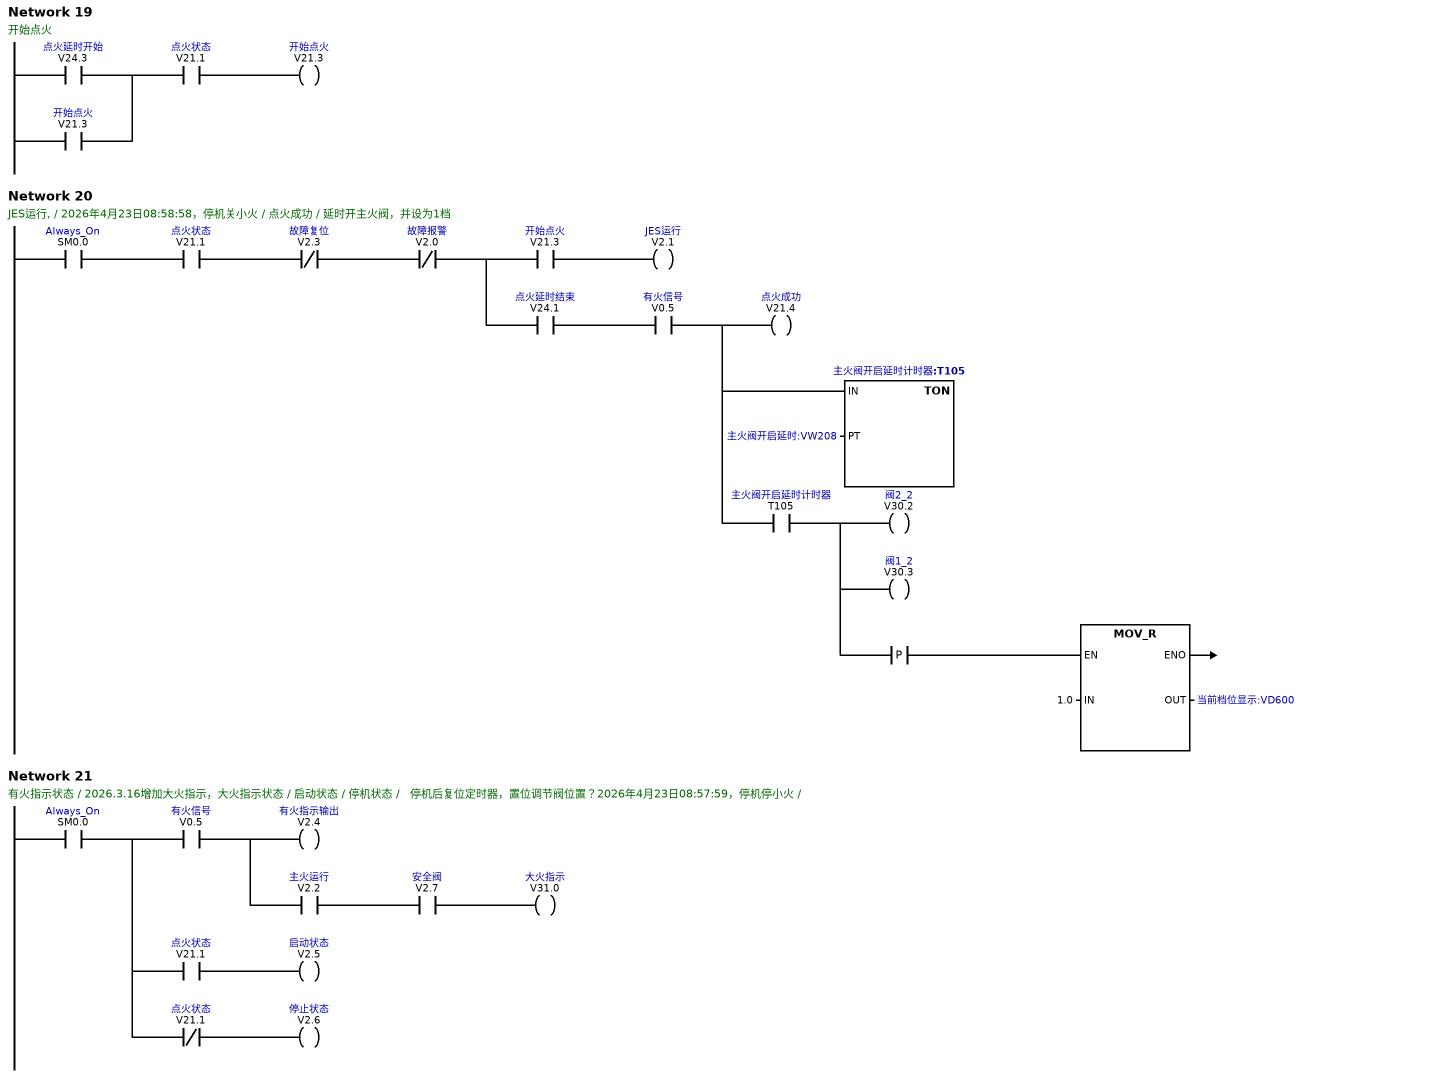
Network 19
// 开始点火
LD     点火延时开始:V24.3
O      开始点火:V21.3
A      点火状态:V21.1
=      开始点火:V21.3
Network 20
// JES运行,
// 2026年4月23日08:58:58，停机关小火
// 点火成功
// 延时开主火阀，并设为1档
LD     Always_On:SM0.0
A      点火状态:V21.1
AN     故障复位:V2.3
AN     故障报警:V2.0
LPS
A      开始点火:V21.3
=      JES运行:V2.1
LPP
A      点火延时结束:V24.1
A      有火信号:V0.5
=      点火成功:V21.4
TON    主火阀开启延时计时器:T105, 主火阀开启延时:VW208
A      主火阀开启延时计时器:T105
=      阀2_2:V30.2
=      阀1_2:V30.3
EU
MOVR   1.0, 当前档位显示:VD600
Network 21
// 有火指示状态
// 2026.3.16增加大火指示，大火指示状态
// 启动状态
// 停机状态
// 	停机后复位定时器，置位调节阀位置？2026年4月23日08:57:59，停机停小火
// 
LD     Always_On:SM0.0
LPS
A      有火信号:V0.5
=      有火指示输出:V2.4
A      主火运行:V2.2
A      安全阀:V2.7
=      大火指示:V31.0
LPP
LPS
A      点火状态:V21.1
=      启动状态:V2.5
LPP
AN     点火状态:V21.1
=      停止状态:V2.6
END_SUBROUTINE_BLOCK

// SBR9: protected block, not included

// SBR10: protected block, not included

SUBROUTINE_BLOCK 手动切档:SBR11
TITLE=
BEGIN
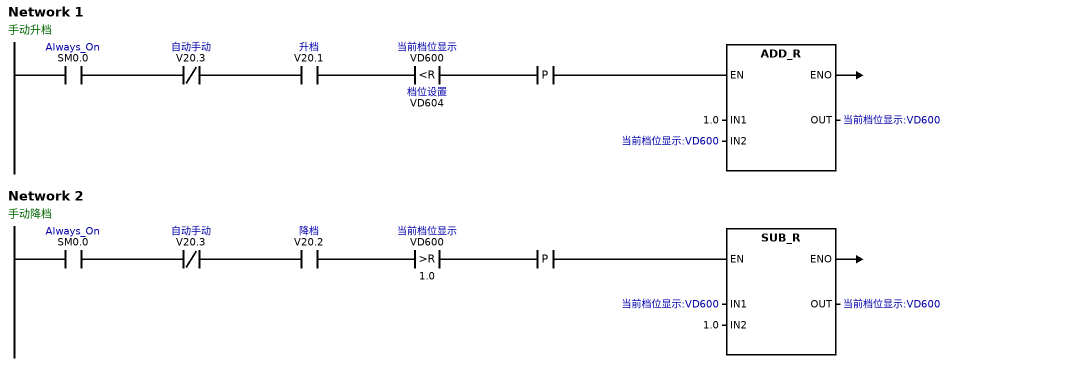
Network 1
// 手动升档
LD     Always_On:SM0.0
AN     自动手动:V20.3
A      升档:V20.1
AR<    当前档位显示:VD600, 档位设置:VD604
EU
+R     1.0, 当前档位显示:VD600
Network 2
// 手动降档
LD     Always_On:SM0.0
AN     自动手动:V20.3
A      降档:V20.2
AR>    当前档位显示:VD600, 1.0
EU
-R     1.0, 当前档位显示:VD600
END_SUBROUTINE_BLOCK

SUBROUTINE_BLOCK 开度档位处理:SBR12
TITLE=
BEGIN
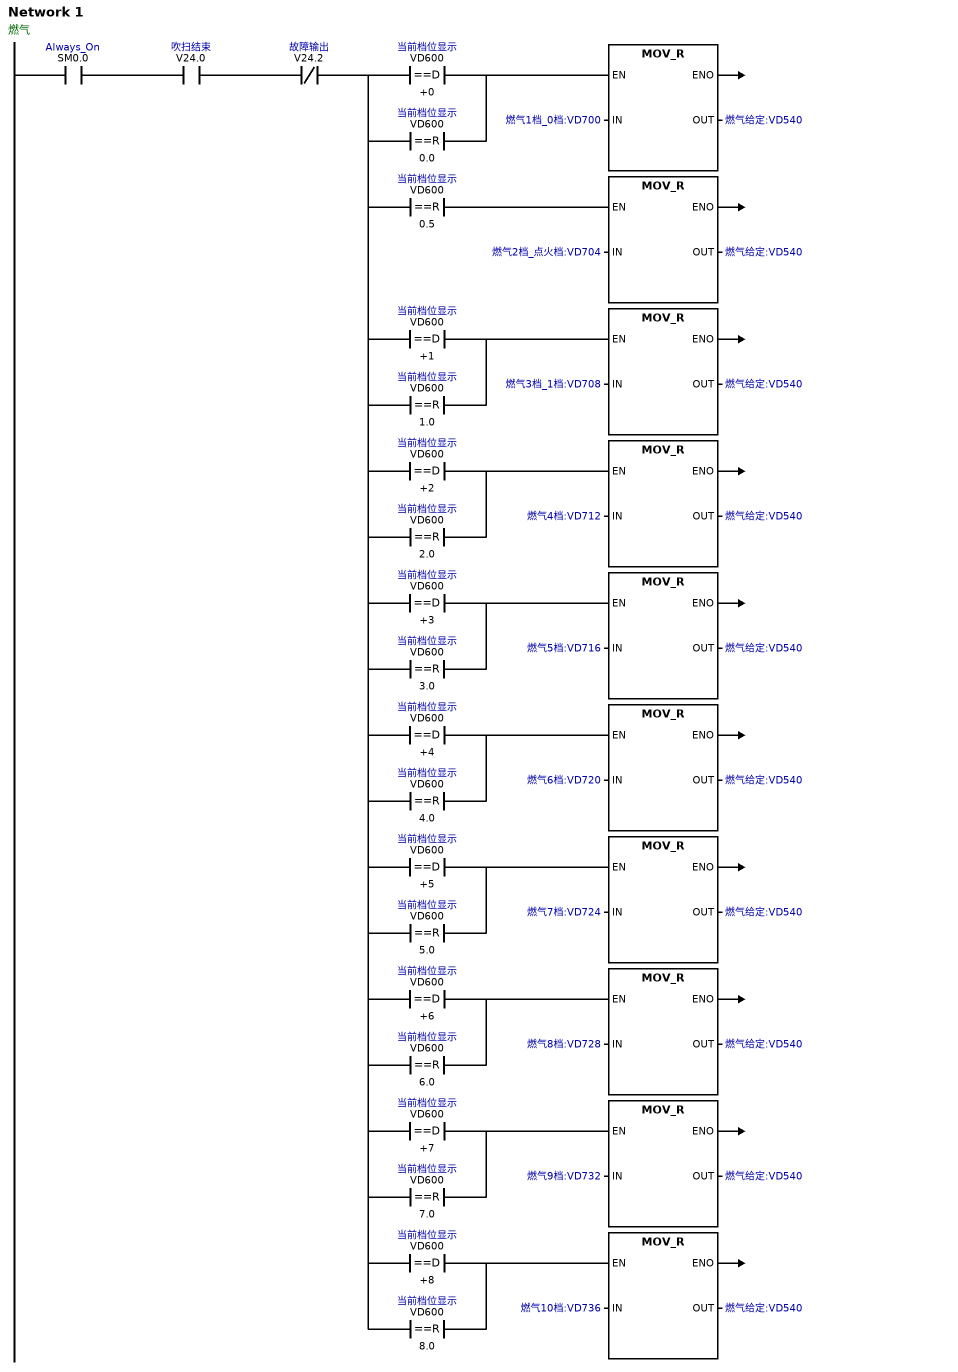
Network 1
// 燃气
LD     Always_On:SM0.0
A      吹扫结束:V24.0
AN     故障输出:V24.2
LPS
LDD=   当前档位显示:VD600, +0
OR=    当前档位显示:VD600, 0.0
ALD
MOVR   燃气1档_0档:VD700, 燃气给定:VD540
LRD
AR=    当前档位显示:VD600, 0.5
MOVR   燃气2档_点火档:VD704, 燃气给定:VD540
LRD
LDD=   当前档位显示:VD600, +1
OR=    当前档位显示:VD600, 1.0
ALD
MOVR   燃气3档_1档:VD708, 燃气给定:VD540
LRD
LDD=   当前档位显示:VD600, +2
OR=    当前档位显示:VD600, 2.0
ALD
MOVR   燃气4档:VD712, 燃气给定:VD540
LRD
LDD=   当前档位显示:VD600, +3
OR=    当前档位显示:VD600, 3.0
ALD
MOVR   燃气5档:VD716, 燃气给定:VD540
LRD
LDD=   当前档位显示:VD600, +4
OR=    当前档位显示:VD600, 4.0
ALD
MOVR   燃气6档:VD720, 燃气给定:VD540
LRD
LDD=   当前档位显示:VD600, +5
OR=    当前档位显示:VD600, 5.0
ALD
MOVR   燃气7档:VD724, 燃气给定:VD540
LRD
LDD=   当前档位显示:VD600, +6
OR=    当前档位显示:VD600, 6.0
ALD
MOVR   燃气8档:VD728, 燃气给定:VD540
LRD
LDD=   当前档位显示:VD600, +7
OR=    当前档位显示:VD600, 7.0
ALD
MOVR   燃气9档:VD732, 燃气给定:VD540
LPP
LDD=   当前档位显示:VD600, +8
OR=    当前档位显示:VD600, 8.0
ALD
MOVR   燃气10档:VD736, 燃气给定:VD540
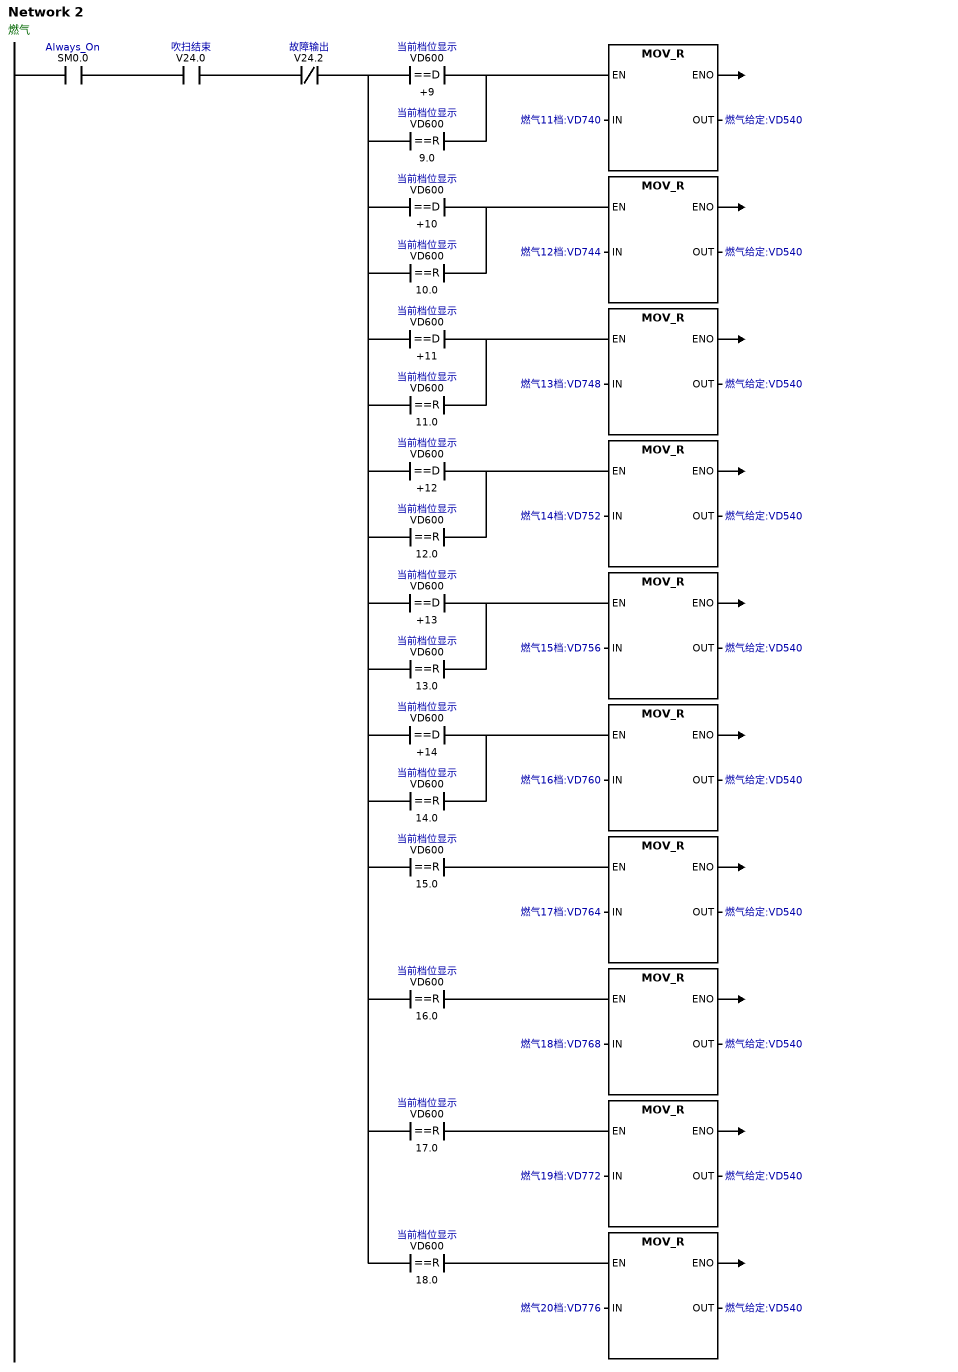
Network 2
// 燃气
LD     Always_On:SM0.0
A      吹扫结束:V24.0
AN     故障输出:V24.2
LPS
LDD=   当前档位显示:VD600, +9
OR=    当前档位显示:VD600, 9.0
ALD
MOVR   燃气11档:VD740, 燃气给定:VD540
LRD
LDD=   当前档位显示:VD600, +10
OR=    当前档位显示:VD600, 10.0
ALD
MOVR   燃气12档:VD744, 燃气给定:VD540
LRD
LDD=   当前档位显示:VD600, +11
OR=    当前档位显示:VD600, 11.0
ALD
MOVR   燃气13档:VD748, 燃气给定:VD540
LRD
LDD=   当前档位显示:VD600, +12
OR=    当前档位显示:VD600, 12.0
ALD
MOVR   燃气14档:VD752, 燃气给定:VD540
LRD
LDD=   当前档位显示:VD600, +13
OR=    当前档位显示:VD600, 13.0
ALD
MOVR   燃气15档:VD756, 燃气给定:VD540
LRD
LDD=   当前档位显示:VD600, +14
OR=    当前档位显示:VD600, 14.0
ALD
MOVR   燃气16档:VD760, 燃气给定:VD540
LPP
LPS
AR=    当前档位显示:VD600, 15.0
MOVR   燃气17档:VD764, 燃气给定:VD540
LRD
AR=    当前档位显示:VD600, 16.0
MOVR   燃气18档:VD768, 燃气给定:VD540
LRD
AR=    当前档位显示:VD600, 17.0
MOVR   燃气19档:VD772, 燃气给定:VD540
LPP
AR=    当前档位显示:VD600, 18.0
MOVR   燃气20档:VD776, 燃气给定:VD540
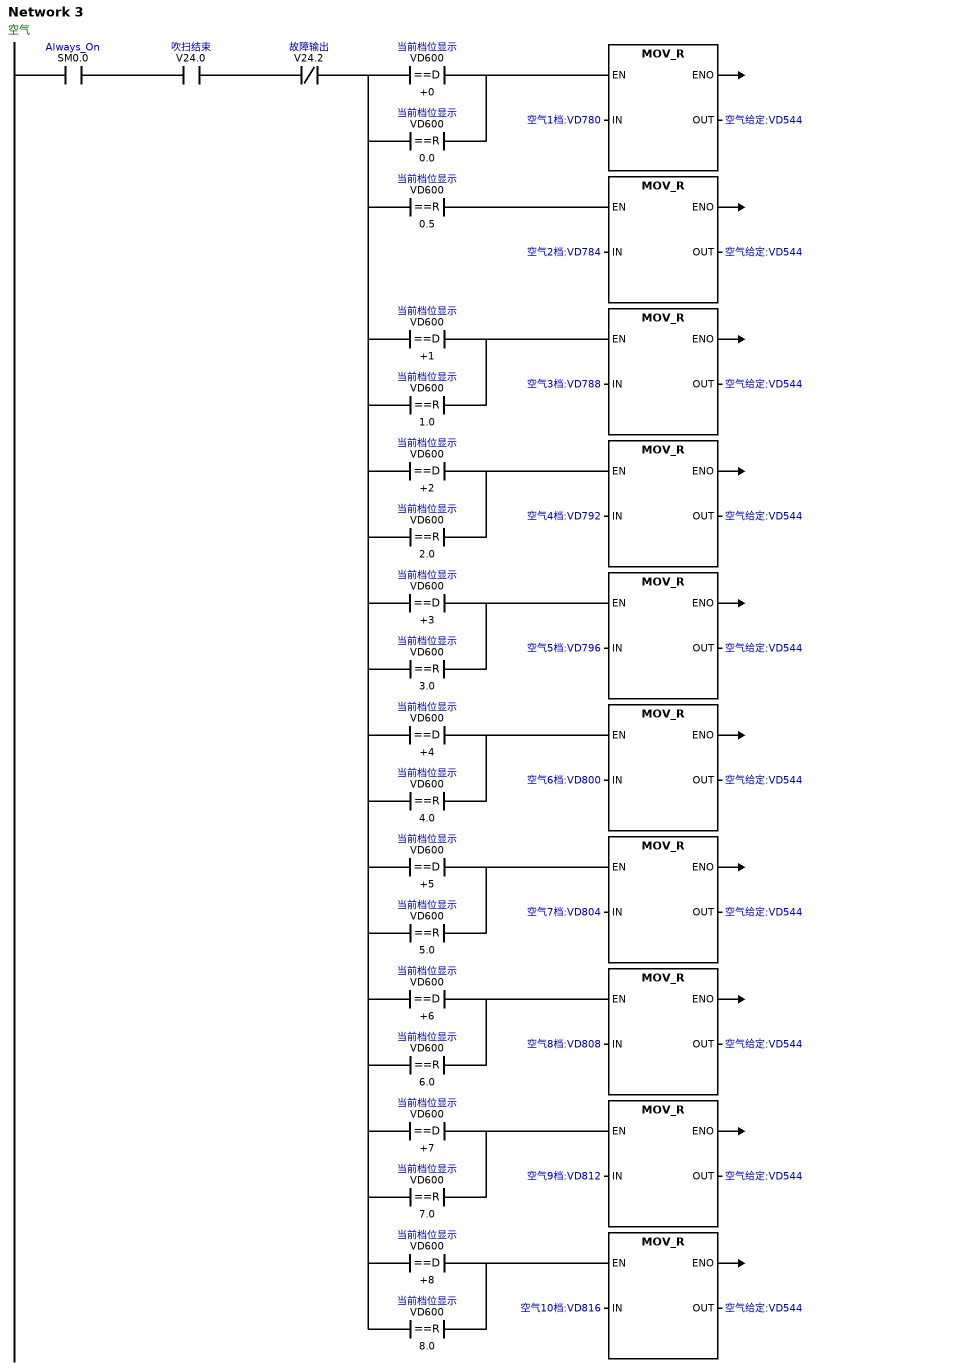
Network 3
// 空气
LD     Always_On:SM0.0
A      吹扫结束:V24.0
AN     故障输出:V24.2
LPS
LDD=   当前档位显示:VD600, +0
OR=    当前档位显示:VD600, 0.0
ALD
MOVR   空气1档:VD780, 空气给定:VD544
LRD
AR=    当前档位显示:VD600, 0.5
MOVR   空气2档:VD784, 空气给定:VD544
LRD
LDD=   当前档位显示:VD600, +1
OR=    当前档位显示:VD600, 1.0
ALD
MOVR   空气3档:VD788, 空气给定:VD544
LRD
LDD=   当前档位显示:VD600, +2
OR=    当前档位显示:VD600, 2.0
ALD
MOVR   空气4档:VD792, 空气给定:VD544
LRD
LDD=   当前档位显示:VD600, +3
OR=    当前档位显示:VD600, 3.0
ALD
MOVR   空气5档:VD796, 空气给定:VD544
LRD
LDD=   当前档位显示:VD600, +4
OR=    当前档位显示:VD600, 4.0
ALD
MOVR   空气6档:VD800, 空气给定:VD544
LRD
LDD=   当前档位显示:VD600, +5
OR=    当前档位显示:VD600, 5.0
ALD
MOVR   空气7档:VD804, 空气给定:VD544
LRD
LDD=   当前档位显示:VD600, +6
OR=    当前档位显示:VD600, 6.0
ALD
MOVR   空气8档:VD808, 空气给定:VD544
LRD
LDD=   当前档位显示:VD600, +7
OR=    当前档位显示:VD600, 7.0
ALD
MOVR   空气9档:VD812, 空气给定:VD544
LPP
LDD=   当前档位显示:VD600, +8
OR=    当前档位显示:VD600, 8.0
ALD
MOVR   空气10档:VD816, 空气给定:VD544
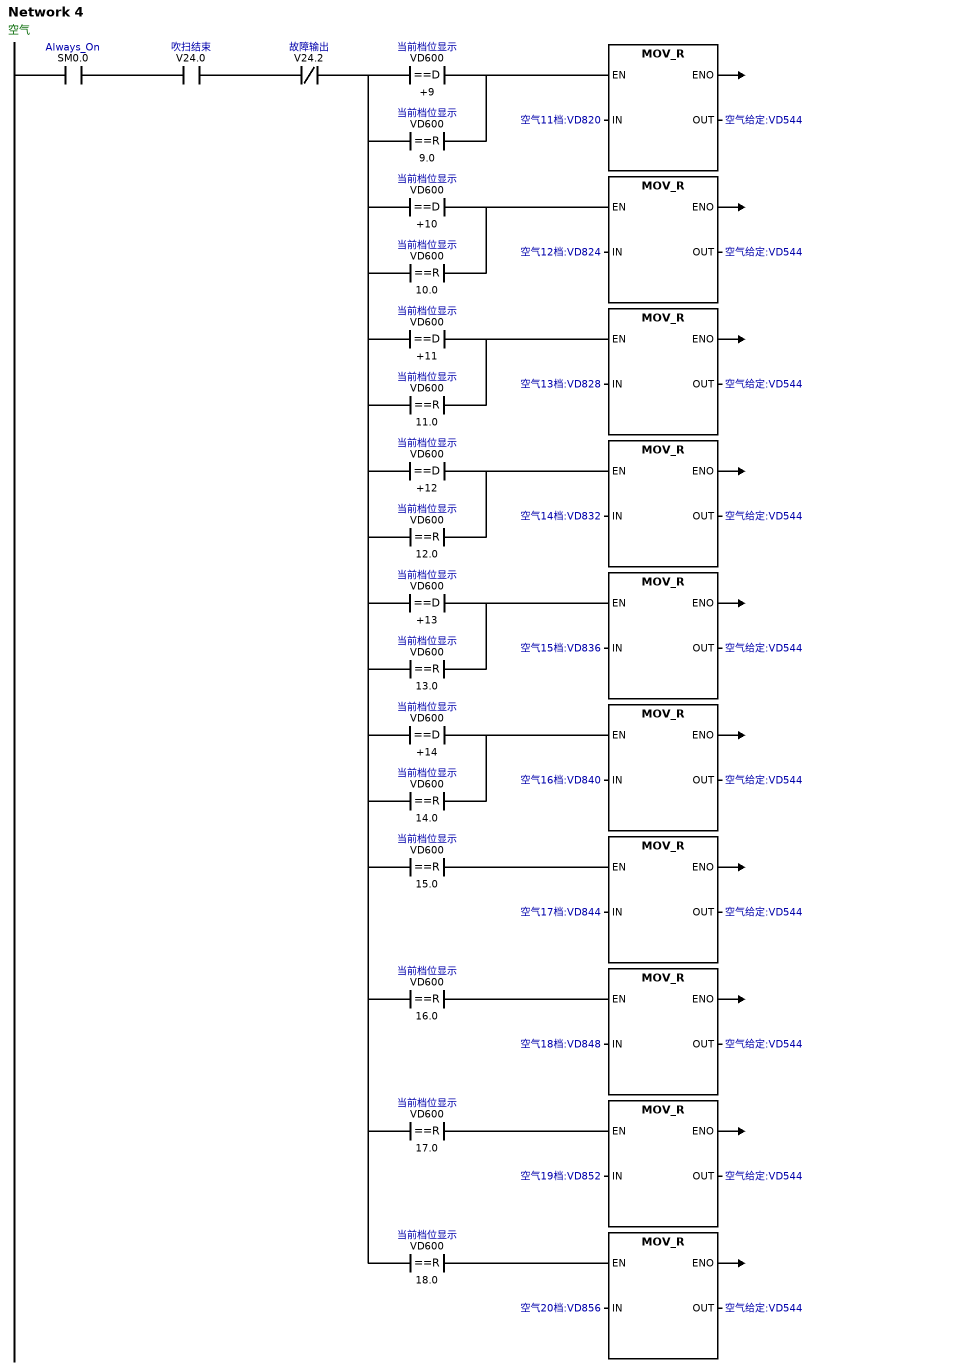
Network 4
// 空气
LD     Always_On:SM0.0
A      吹扫结束:V24.0
AN     故障输出:V24.2
LPS
LDD=   当前档位显示:VD600, +9
OR=    当前档位显示:VD600, 9.0
ALD
MOVR   空气11档:VD820, 空气给定:VD544
LRD
LDD=   当前档位显示:VD600, +10
OR=    当前档位显示:VD600, 10.0
ALD
MOVR   空气12档:VD824, 空气给定:VD544
LRD
LDD=   当前档位显示:VD600, +11
OR=    当前档位显示:VD600, 11.0
ALD
MOVR   空气13档:VD828, 空气给定:VD544
LRD
LDD=   当前档位显示:VD600, +12
OR=    当前档位显示:VD600, 12.0
ALD
MOVR   空气14档:VD832, 空气给定:VD544
LRD
LDD=   当前档位显示:VD600, +13
OR=    当前档位显示:VD600, 13.0
ALD
MOVR   空气15档:VD836, 空气给定:VD544
LRD
LDD=   当前档位显示:VD600, +14
OR=    当前档位显示:VD600, 14.0
ALD
MOVR   空气16档:VD840, 空气给定:VD544
LPP
LPS
AR=    当前档位显示:VD600, 15.0
MOVR   空气17档:VD844, 空气给定:VD544
LRD
AR=    当前档位显示:VD600, 16.0
MOVR   空气18档:VD848, 空气给定:VD544
LRD
AR=    当前档位显示:VD600, 17.0
MOVR   空气19档:VD852, 空气给定:VD544
LPP
AR=    当前档位显示:VD600, 18.0
MOVR   空气20档:VD856, 空气给定:VD544
